TYPE "UDT_VfdSEWPositioningPO"
TITLE = UDT_VFD_SEW_PO
VERSION : 0.1
//User-defined structure of VFD SEW output telegram.
   STRUCT
      Control_Word_1 : Struct   // Control Word 1
         ResetError { ExternalAccessible := 'False'; ExternalVisible := 'False'; ExternalWritable := 'False'} : Bool;   // Reset error "1"
         BIT_09_Reserved { ExternalAccessible := 'False'; ExternalVisible := 'False'; ExternalWritable := 'False'} : Bool;   // Reserved
         ActivateDriveTrain2 { ExternalAccessible := 'False'; ExternalVisible := 'False'; ExternalWritable := 'False'} : Bool;   // Activate drive train 2 "1"
         BIT_11_Reserved { ExternalAccessible := 'False'; ExternalVisible := 'False'; ExternalWritable := 'False'} : Bool;   // Reserved
         DeactivateSW_LimitSwitch { ExternalAccessible := 'False'; ExternalVisible := 'False'; ExternalWritable := 'False'} : Bool;   // Deactivate software limit switch "1"
         ActivateInhibit { ExternalAccessible := 'False'; ExternalVisible := 'False'; ExternalWritable := 'False'} : Bool;   // Activate inhibit "1"
         ActivateStandby { ExternalAccessible := 'False'; ExternalVisible := 'False'; ExternalWritable := 'False'} : Bool;   // Activate standby "1"
         MovikitHandshakeIn { ExternalAccessible := 'False'; ExternalVisible := 'False'; ExternalWritable := 'False'} : Bool;   // If the MOVIKIT works the value will be copied into "MovikitHandshakeOut"
         EnableRapidStop { ExternalAccessible := 'False'; ExternalVisible := 'False'; ExternalWritable := 'False'} : Bool;   // Enable “1” / Rapid stop “0”
         EnableApplicationStop { ExternalAccessible := 'False'; ExternalVisible := 'False'; ExternalWritable := 'False'} : Bool;   // Enable “1” / Application stop “0”
         BIT_02_Reserved { ExternalAccessible := 'False'; ExternalVisible := 'False'; ExternalWritable := 'False'} : Bool;   // Reserved
         ReleaseBrake { ExternalAccessible := 'False'; ExternalVisible := 'False'; ExternalWritable := 'False'} : Bool;   // Release brake "1"
         JogPos { ExternalAccessible := 'False'; ExternalVisible := 'False'; ExternalWritable := 'False'} : Bool;   // Jog in positive direction "1"
         JogNeg { ExternalAccessible := 'False'; ExternalVisible := 'False'; ExternalWritable := 'False'} : Bool;   // Jog in negative direction "1"
         ApplyRelativePositioning { ExternalAccessible := 'False'; ExternalVisible := 'False'; ExternalWritable := 'False'} : Bool;   // Take the relative position from the FCB09 "1"
         StartStop { ExternalAccessible := 'False'; ExternalVisible := 'False'; ExternalWritable := 'False'} : Bool;   // Start "1" / Stop "0"
      END_STRUCT;
      SetpointSpeed : Int;   // Speed (Int) [mm/s]
      SetpointAcceleration : Int;   // Acceleration (Int) [mm/s²]
      SetpointDeceleration : Int;   // Decceleration (Int) [mm/s²]
      DigitalOutputs : Word;   // Digital Outputs
      SetpointMode : Int;   // Set the application mode (Int)
      SetpointPosition_hW : Word;   // Setpoint Position - High Word
      SetpointPosition_lW : Word;   // Setpoint Position - Low Word
   END_STRUCT;

END_TYPE

TYPE "UDT_Message"
TITLE = UDT_Message
VERSION : 0.1
//User-defined structure of the message characters array.
   STRUCT
      Character : Array[0..499] of Char;   // Message character
   END_STRUCT;

END_TYPE

TYPE "UDT_TCPIPReceiveStatistics"
TITLE = UDT_TCPIPReceiveStatistics
VERSION : 0.1
//User-defined structure of FB_TCPIPReceive function block statistics.
   STRUCT
      InvalidMsg : UInt;   // Invalid message received
   END_STRUCT;

END_TYPE

TYPE "UDT_SystemStatistics"
TITLE = Cabinet MCP Statistics
VERSION : 0.1
   STRUCT
      HMI_Stop : "UDT_EventStatistic";   // HMI stop statistics
      Field_Stop : "UDT_EventStatistic";   // Field stop statistics
      Building_EStop : "UDT_EventStatistic";   // Bulding emergency stop statistics
      MCP_EStop : "UDT_EventStatistic";   // MCP emergency stop statistics
      RemotePanel_EStop : "UDT_EventStatistic";   // Remote panel emergency stop statistics
      Error : "UDT_EventStatistic";   // System in error
      StartNumberOfTimes { S7_SetPoint := 'True'} : DInt;   // Number of times system started
      ResetNumberOfTimes { S7_SetPoint := 'True'} : DInt;   // Number of timer system reset
      DataResetNumberOfTimes { S7_SetPoint := 'True'} : DInt;   // Number of data reset
   END_STRUCT;

END_TYPE

TYPE "UDT_ProfiDiagStatistics"
TITLE = UDT_ProfiDiagStatistics
VERSION : 0.1
//User-defined structure of FB_ProfiDiag function block statistics.
   STRUCT
      DeviceError { S7_SetPoint := 'False'} : Array[0..512] of "UDT_EventStatistic";   // Device error statistics
   END_STRUCT;

END_TYPE

TYPE "UDT_PowerDistributionPanelCBState"
VERSION : 0.1
   STRUCT
      CircuitBreakerStateF100 { ExternalAccessible := 'False'; ExternalVisible := 'False'; ExternalWritable := 'False'} : Bool;   // Circuit Breaker State Ok if the signal is true
      CircuitBreakerStateF201 { ExternalAccessible := 'False'; ExternalVisible := 'False'; ExternalWritable := 'False'} : Bool;   // Circuit Breaker State Ok if the signal is true
      CircuitBreakerStateF202 { ExternalAccessible := 'False'; ExternalVisible := 'False'; ExternalWritable := 'False'} : Bool;   // Circuit Breaker State Ok if the signal is true
      CircuitBreakerStateF203 { ExternalAccessible := 'False'; ExternalVisible := 'False'; ExternalWritable := 'False'} : Bool;   // Circuit Breaker State Ok if the signal is true
      CircuitBreakerStateF204 { ExternalAccessible := 'False'; ExternalVisible := 'False'; ExternalWritable := 'False'} : Bool;   // Circuit Breaker State Ok if the signal is true
      CircuitBreakerStateF205 { ExternalAccessible := 'False'; ExternalVisible := 'False'; ExternalWritable := 'False'} : Bool;   // Circuit Breaker State Ok if the signal is true
      CircuitBreakerStateF206 { ExternalAccessible := 'False'; ExternalVisible := 'False'; ExternalWritable := 'False'} : Bool;   // Circuit Breaker State Ok if the signal is true
      CircuitBreakerStateF207 { ExternalAccessible := 'False'; ExternalVisible := 'False'; ExternalWritable := 'False'} : Bool;   // Circuit Breaker State Ok if the signal is true
      CircuitBreakerStateF208 { ExternalAccessible := 'False'; ExternalVisible := 'False'; ExternalWritable := 'False'} : Bool;   // Circuit Breaker State Ok if the signal is true
      CircuitBreakerStateF209 { ExternalAccessible := 'False'; ExternalVisible := 'False'; ExternalWritable := 'False'} : Bool;   // Circuit Breaker State Ok if the signal is true
      CircuitBreakerStateF210 { ExternalAccessible := 'False'; ExternalVisible := 'False'; ExternalWritable := 'False'} : Bool;   // Circuit Breaker State Ok if the signal is true
      CircuitBreakerStateF211 { ExternalAccessible := 'False'; ExternalVisible := 'False'; ExternalWritable := 'False'} : Bool;   // Circuit Breaker State Ok if the signal is true
      CircuitBreakerStateF212 { ExternalAccessible := 'False'; ExternalVisible := 'False'; ExternalWritable := 'False'} : Bool;   // Circuit Breaker State Ok if the signal is true
      CircuitBreakerStateF213 { ExternalAccessible := 'False'; ExternalVisible := 'False'; ExternalWritable := 'False'} : Bool;   // Circuit Breaker State Ok if the signal is true
      CircuitBreakerStateF214 { ExternalAccessible := 'False'; ExternalVisible := 'False'; ExternalWritable := 'False'} : Bool;   // Circuit Breaker State Ok if the signal is true
      CircuitBreakerStateF215 { ExternalAccessible := 'False'; ExternalVisible := 'False'; ExternalWritable := 'False'} : Bool;   // Circuit Breaker State Ok if the signal is true
      CircuitBreakerStateF216 { ExternalAccessible := 'False'; ExternalVisible := 'False'; ExternalWritable := 'False'} : Bool;   // Circuit Breaker State Ok if the signal is true
      CircuitBreakerStateF217 { ExternalAccessible := 'False'; ExternalVisible := 'False'; ExternalWritable := 'False'} : Bool;   // Circuit Breaker State Ok if the signal is true
      CircuitBreakerStateF218 { ExternalAccessible := 'False'; ExternalVisible := 'False'; ExternalWritable := 'False'} : Bool;   // Circuit Breaker State Ok if the signal is true
      CircuitBreakerStateF219 { ExternalAccessible := 'False'; ExternalVisible := 'False'; ExternalWritable := 'False'} : Bool;   // Circuit Breaker State Ok if the signal is true
      CircuitBreakerStateF220 { ExternalAccessible := 'False'; ExternalVisible := 'False'; ExternalWritable := 'False'} : Bool;   // Circuit Breaker State Ok if the signal is true
      CircuitBreakerStateF221 { ExternalAccessible := 'False'; ExternalVisible := 'False'; ExternalWritable := 'False'} : Bool;   // Circuit Breaker State Ok if the signal is true
      CircuitBreakerStateF222 { ExternalAccessible := 'False'; ExternalVisible := 'False'; ExternalWritable := 'False'} : Bool;   // Circuit Breaker State Ok if the signal is true
      CircuitBreakerStateF223 { ExternalAccessible := 'False'; ExternalVisible := 'False'; ExternalWritable := 'False'} : Bool;   // Circuit Breaker State Ok if the signal is true
      CircuitBreakerStateF224 { ExternalAccessible := 'False'; ExternalVisible := 'False'; ExternalWritable := 'False'} : Bool;   // Circuit Breaker State Ok if the signal is true
      CircuitBreakerStateF225 { ExternalAccessible := 'False'; ExternalVisible := 'False'; ExternalWritable := 'False'} : Bool;   // Circuit Breaker State Ok if the signal is true
      CircuitBreakerStateF226 { ExternalAccessible := 'False'; ExternalVisible := 'False'; ExternalWritable := 'False'} : Bool;   // Circuit Breaker State Ok if the signal is true
      CircuitBreakerStateF227 { ExternalAccessible := 'False'; ExternalVisible := 'False'; ExternalWritable := 'False'} : Bool;   // Circuit Breaker State Ok if the signal is true
      CircuitBreakerStateF228 { ExternalAccessible := 'False'; ExternalVisible := 'False'; ExternalWritable := 'False'} : Bool;   // Circuit Breaker State Ok if the signal is true
      CircuitBreakerStateF229 { ExternalAccessible := 'False'; ExternalVisible := 'False'; ExternalWritable := 'False'} : Bool;   // Circuit Breaker State Ok if the signal is true
      CircuitBreakerStateF230 { ExternalAccessible := 'False'; ExternalVisible := 'False'; ExternalWritable := 'False'} : Bool;   // Circuit Breaker State Ok if the signal is true
      CircuitBreakerStateF231 { ExternalAccessible := 'False'; ExternalVisible := 'False'; ExternalWritable := 'False'} : Bool;   // Circuit Breaker State Ok if the signal is true
      CircuitBreakerStateF232 { ExternalAccessible := 'False'; ExternalVisible := 'False'; ExternalWritable := 'False'} : Bool;   // Circuit Breaker State Ok if the signal is true
      CircuitBreakerStateF233 { ExternalAccessible := 'False'; ExternalVisible := 'False'; ExternalWritable := 'False'} : Bool;   // Circuit Breaker State Ok if the signal is true
      CircuitBreakerStateF234 { ExternalAccessible := 'False'; ExternalVisible := 'False'; ExternalWritable := 'False'} : Bool;   // Circuit Breaker State Ok if the signal is true
      CircuitBreakerStateF235 { ExternalAccessible := 'False'; ExternalVisible := 'False'; ExternalWritable := 'False'} : Bool;   // Circuit Breaker State Ok if the signal is true
      CircuitBreakerStateF236 { ExternalAccessible := 'False'; ExternalVisible := 'False'; ExternalWritable := 'False'} : Bool;   // Circuit Breaker State Ok if the signal is true
      CircuitBreakerStateF237 { ExternalAccessible := 'False'; ExternalVisible := 'False'; ExternalWritable := 'False'} : Bool;   // Circuit Breaker State Ok if the signal is true
      CircuitBreakerStateF238 { ExternalAccessible := 'False'; ExternalVisible := 'False'; ExternalWritable := 'False'} : Bool;   // Circuit Breaker State Ok if the signal is true
      CircuitBreakerStateF239 { ExternalAccessible := 'False'; ExternalVisible := 'False'; ExternalWritable := 'False'} : Bool;   // Circuit Breaker State Ok if the signal is true
      CircuitBreakerStateF240 { ExternalAccessible := 'False'; ExternalVisible := 'False'; ExternalWritable := 'False'} : Bool;   // Circuit Breaker State Ok if the signal is true
      CircuitBreakerStateF241 { ExternalAccessible := 'False'; ExternalVisible := 'False'; ExternalWritable := 'False'} : Bool;   // Circuit Breaker State Ok if the signal is true
      CircuitBreakerStateF242 { ExternalAccessible := 'False'; ExternalVisible := 'False'; ExternalWritable := 'False'} : Bool;   // Circuit Breaker State Ok if the signal is true
      CircuitBreakerStateF243 { ExternalAccessible := 'False'; ExternalVisible := 'False'; ExternalWritable := 'False'} : Bool;   // Circuit Breaker State Ok if the signal is true
      CircuitBreakerStateF244 { ExternalAccessible := 'False'; ExternalVisible := 'False'; ExternalWritable := 'False'} : Bool;   // Circuit Breaker State Ok if the signal is true
      CircuitBreakerStateF245 { ExternalAccessible := 'False'; ExternalVisible := 'False'; ExternalWritable := 'False'} : Bool;   // Circuit Breaker State Ok if the signal is true
      CircuitBreakerStateF246 { ExternalAccessible := 'False'; ExternalVisible := 'False'; ExternalWritable := 'False'} : Bool;   // Circuit Breaker State Ok if the signal is true
      CircuitBreakerStateF247 { ExternalAccessible := 'False'; ExternalVisible := 'False'; ExternalWritable := 'False'} : Bool;   // Circuit Breaker State Ok if the signal is true
      CircuitBreakerStateF248 { ExternalAccessible := 'False'; ExternalVisible := 'False'; ExternalWritable := 'False'} : Bool;   // Circuit Breaker State Ok if the signal is true
      CircuitBreakerStateF249 { ExternalAccessible := 'False'; ExternalVisible := 'False'; ExternalWritable := 'False'} : Bool;   // Circuit Breaker State Ok if the signal is true
      CircuitBreakerStateF250 { ExternalAccessible := 'False'; ExternalVisible := 'False'; ExternalWritable := 'False'} : Bool;   // Circuit Breaker State Ok if the signal is true
      CircuitBreakerStateF251 { ExternalAccessible := 'False'; ExternalVisible := 'False'; ExternalWritable := 'False'} : Bool;   // Circuit Breaker State Ok if the signal is true
      CircuitBreakerStateF501 { ExternalAccessible := 'False'; ExternalVisible := 'False'; ExternalWritable := 'False'} : Bool;   // Circuit Breaker State Ok if the signal is true
      CircuitBreakerStateF502 { ExternalAccessible := 'False'; ExternalVisible := 'False'; ExternalWritable := 'False'} : Bool;   // Circuit Breaker State Ok if the signal is true
      CircuitBreakerStateF503 { ExternalAccessible := 'False'; ExternalVisible := 'False'; ExternalWritable := 'False'} : Bool;   // Circuit Breaker State Ok if the signal is true
      CircuitBreakerStateF504 { ExternalAccessible := 'False'; ExternalVisible := 'False'; ExternalWritable := 'False'} : Bool;   // Circuit Breaker State Ok if the signal is true
      CircuitBreakerStateF505 { ExternalAccessible := 'False'; ExternalVisible := 'False'; ExternalWritable := 'False'} : Bool;   // Circuit Breaker State Ok if the signal is true
   END_STRUCT;

END_TYPE

TYPE "UDT_PowerDistributionPanelStatus"
VERSION : 0.1
   STRUCT
      Status : Int;   // Status number
      Specific : Struct
         CircuitBreakersTripped { ExternalAccessible := 'False'; ExternalVisible := 'False'; ExternalWritable := 'False'} : Bool;   // Circuit breakers tripped when the value is true
         CircuitBreakerTrippedF100 { ExternalAccessible := 'False'; ExternalVisible := 'False'; ExternalWritable := 'False'} : Bool;   // Circuit breaker is tripped when the value is true
         CircuitBreakerTrippedF201 { ExternalAccessible := 'False'; ExternalVisible := 'False'; ExternalWritable := 'False'} : Bool;   // Circuit breaker is tripped when the value is true
         CircuitBreakerTrippedF202 { ExternalAccessible := 'False'; ExternalVisible := 'False'; ExternalWritable := 'False'} : Bool;   // Circuit breaker is tripped when the value is true
         CircuitBreakerTrippedF203 { ExternalAccessible := 'False'; ExternalVisible := 'False'; ExternalWritable := 'False'} : Bool;   // Circuit breaker is tripped when the value is true
         CircuitBreakerTrippedF204 { ExternalAccessible := 'False'; ExternalVisible := 'False'; ExternalWritable := 'False'} : Bool;   // Circuit breaker is tripped when the value is true
         CircuitBreakerTrippedF205 { ExternalAccessible := 'False'; ExternalVisible := 'False'; ExternalWritable := 'False'} : Bool;   // Circuit breaker is tripped when the value is true
         CircuitBreakerTrippedF206 { ExternalAccessible := 'False'; ExternalVisible := 'False'; ExternalWritable := 'False'} : Bool;   // Circuit breaker is tripped when the value is true
         CircuitBreakerTrippedF207 { ExternalAccessible := 'False'; ExternalVisible := 'False'; ExternalWritable := 'False'} : Bool;   // Circuit breaker is tripped when the value is true
         CircuitBreakerTrippedF208 { ExternalAccessible := 'False'; ExternalVisible := 'False'; ExternalWritable := 'False'} : Bool;   // Circuit breaker is tripped when the value is true
         CircuitBreakerTrippedF209 { ExternalAccessible := 'False'; ExternalVisible := 'False'; ExternalWritable := 'False'} : Bool;   // Circuit breaker is tripped when the value is true
         CircuitBreakerTrippedF210 { ExternalAccessible := 'False'; ExternalVisible := 'False'; ExternalWritable := 'False'} : Bool;   // Circuit breaker is tripped when the value is true
         CircuitBreakerTrippedF211 { ExternalAccessible := 'False'; ExternalVisible := 'False'; ExternalWritable := 'False'} : Bool;   // Circuit breaker is tripped when the value is true
         CircuitBreakerTrippedF212 { ExternalAccessible := 'False'; ExternalVisible := 'False'; ExternalWritable := 'False'} : Bool;   // Circuit breaker is tripped when the value is true
         CircuitBreakerTrippedF213 { ExternalAccessible := 'False'; ExternalVisible := 'False'; ExternalWritable := 'False'} : Bool;   // Circuit breaker is tripped when the value is true
         CircuitBreakerTrippedF214 { ExternalAccessible := 'False'; ExternalVisible := 'False'; ExternalWritable := 'False'} : Bool;   // Circuit breaker is tripped when the value is true
         CircuitBreakerTrippedF215 { ExternalAccessible := 'False'; ExternalVisible := 'False'; ExternalWritable := 'False'} : Bool;   // Circuit breaker is tripped when the value is true
         CircuitBreakerTrippedF216 { ExternalAccessible := 'False'; ExternalVisible := 'False'; ExternalWritable := 'False'} : Bool;   // Circuit breaker is tripped when the value is true
         CircuitBreakerTrippedF217 { ExternalAccessible := 'False'; ExternalVisible := 'False'; ExternalWritable := 'False'} : Bool;   // Circuit breaker is tripped when the value is true
         CircuitBreakerTrippedF218 { ExternalAccessible := 'False'; ExternalVisible := 'False'; ExternalWritable := 'False'} : Bool;   // Circuit breaker is tripped when the value is true
         CircuitBreakerTrippedF219 { ExternalAccessible := 'False'; ExternalVisible := 'False'; ExternalWritable := 'False'} : Bool;   // Circuit breaker is tripped when the value is true
         CircuitBreakerTrippedF220 { ExternalAccessible := 'False'; ExternalVisible := 'False'; ExternalWritable := 'False'} : Bool;   // Circuit breaker is tripped when the value is true
         CircuitBreakerTrippedF221 { ExternalAccessible := 'False'; ExternalVisible := 'False'; ExternalWritable := 'False'} : Bool;   // Circuit breaker is tripped when the value is true
         CircuitBreakerTrippedF222 { ExternalAccessible := 'False'; ExternalVisible := 'False'; ExternalWritable := 'False'} : Bool;   // Circuit breaker is tripped when the value is true
         CircuitBreakerTrippedF223 { ExternalAccessible := 'False'; ExternalVisible := 'False'; ExternalWritable := 'False'} : Bool;   // Circuit breaker is tripped when the value is true
         CircuitBreakerTrippedF224 { ExternalAccessible := 'False'; ExternalVisible := 'False'; ExternalWritable := 'False'} : Bool;   // Circuit breaker is tripped when the value is true
         CircuitBreakerTrippedF225 { ExternalAccessible := 'False'; ExternalVisible := 'False'; ExternalWritable := 'False'} : Bool;   // Circuit breaker is tripped when the value is true
         CircuitBreakerTrippedF226 { ExternalAccessible := 'False'; ExternalVisible := 'False'; ExternalWritable := 'False'} : Bool;   // Circuit breaker is tripped when the value is true
         CircuitBreakerTrippedF227 { ExternalAccessible := 'False'; ExternalVisible := 'False'; ExternalWritable := 'False'} : Bool;   // Circuit breaker is tripped when the value is true
         CircuitBreakerTrippedF228 { ExternalAccessible := 'False'; ExternalVisible := 'False'; ExternalWritable := 'False'} : Bool;   // Circuit breaker is tripped when the value is true
         CircuitBreakerTrippedF229 { ExternalAccessible := 'False'; ExternalVisible := 'False'; ExternalWritable := 'False'} : Bool;   // Circuit breaker is tripped when the value is true
         CircuitBreakerTrippedF230 { ExternalAccessible := 'False'; ExternalVisible := 'False'; ExternalWritable := 'False'} : Bool;   // Circuit breaker is tripped when the value is true
         CircuitBreakerTrippedF231 { ExternalAccessible := 'False'; ExternalVisible := 'False'; ExternalWritable := 'False'} : Bool;   // Circuit breaker is tripped when the value is true
         CircuitBreakerTrippedF232 { ExternalAccessible := 'False'; ExternalVisible := 'False'; ExternalWritable := 'False'} : Bool;   // Circuit breaker is tripped when the value is true
         CircuitBreakerTrippedF233 { ExternalAccessible := 'False'; ExternalVisible := 'False'; ExternalWritable := 'False'} : Bool;   // Circuit breaker is tripped when the value is true
         CircuitBreakerTrippedF234 { ExternalAccessible := 'False'; ExternalVisible := 'False'; ExternalWritable := 'False'} : Bool;   // Circuit breaker is tripped when the value is true
         CircuitBreakerTrippedF235 { ExternalAccessible := 'False'; ExternalVisible := 'False'; ExternalWritable := 'False'} : Bool;   // Circuit breaker is tripped when the value is true
         CircuitBreakerTrippedF236 { ExternalAccessible := 'False'; ExternalVisible := 'False'; ExternalWritable := 'False'} : Bool;   // Circuit breaker is tripped when the value is true
         CircuitBreakerTrippedF237 { ExternalAccessible := 'False'; ExternalVisible := 'False'; ExternalWritable := 'False'} : Bool;   // Circuit breaker is tripped when the value is true
         CircuitBreakerTrippedF238 { ExternalAccessible := 'False'; ExternalVisible := 'False'; ExternalWritable := 'False'} : Bool;   // Circuit breaker is tripped when the value is true
         CircuitBreakerTrippedF239 { ExternalAccessible := 'False'; ExternalVisible := 'False'; ExternalWritable := 'False'} : Bool;   // Circuit breaker is tripped when the value is true
         CircuitBreakerTrippedF240 { ExternalAccessible := 'False'; ExternalVisible := 'False'; ExternalWritable := 'False'} : Bool;   // Circuit breaker is tripped when the value is true
         CircuitBreakerTrippedF241 { ExternalAccessible := 'False'; ExternalVisible := 'False'; ExternalWritable := 'False'} : Bool;   // Circuit breaker is tripped when the value is true
         CircuitBreakerTrippedF242 { ExternalAccessible := 'False'; ExternalVisible := 'False'; ExternalWritable := 'False'} : Bool;   // Circuit breaker is tripped when the value is true
         CircuitBreakerTrippedF243 { ExternalAccessible := 'False'; ExternalVisible := 'False'; ExternalWritable := 'False'} : Bool;   // Circuit breaker is tripped when the value is true
         CircuitBreakerTrippedF244 { ExternalAccessible := 'False'; ExternalVisible := 'False'; ExternalWritable := 'False'} : Bool;   // Circuit breaker is tripped when the value is true
         CircuitBreakerTrippedF245 { ExternalAccessible := 'False'; ExternalVisible := 'False'; ExternalWritable := 'False'} : Bool;   // Circuit breaker is tripped when the value is true
         CircuitBreakerTrippedF246 { ExternalAccessible := 'False'; ExternalVisible := 'False'; ExternalWritable := 'False'} : Bool;   // Circuit breaker is tripped when the value is true
         CircuitBreakerTrippedF247 { ExternalAccessible := 'False'; ExternalVisible := 'False'; ExternalWritable := 'False'} : Bool;   // Circuit breaker is tripped when the value is true
         CircuitBreakerTrippedF248 { ExternalAccessible := 'False'; ExternalVisible := 'False'; ExternalWritable := 'False'} : Bool;   // Circuit breaker is tripped when the value is true
         CircuitBreakerTrippedF249 { ExternalAccessible := 'False'; ExternalVisible := 'False'; ExternalWritable := 'False'} : Bool;   // Circuit breaker is tripped when the value is true
         CircuitBreakerTrippedF250 { ExternalAccessible := 'False'; ExternalVisible := 'False'; ExternalWritable := 'False'} : Bool;   // Circuit breaker is tripped when the value is true
         CircuitBreakerTrippedF501 { ExternalAccessible := 'False'; ExternalVisible := 'False'; ExternalWritable := 'False'} : Bool;   // Circuit breaker is tripped when the value is true
         CircuitBreakerTrippedF502 { ExternalAccessible := 'False'; ExternalVisible := 'False'; ExternalWritable := 'False'} : Bool;   // Circuit breaker is tripped when the value is true
         CircuitBreakerTrippedF503 { ExternalAccessible := 'False'; ExternalVisible := 'False'; ExternalWritable := 'False'} : Bool;   // Circuit breaker is tripped when the value is true
         CircuitBreakerTrippedF504 { ExternalAccessible := 'False'; ExternalVisible := 'False'; ExternalWritable := 'False'} : Bool;   // Circuit breaker is tripped when the value is true
         CircuitBreakerTrippedF505 { ExternalAccessible := 'False'; ExternalVisible := 'False'; ExternalWritable := 'False'} : Bool;   // Circuit breaker is tripped when the value is true
      END_STRUCT;
   END_STRUCT;

END_TYPE

TYPE "UDT_XBSInductInterfaceRcv"
VERSION : 0.1
   STRUCT
      Watchdog : Byte;   // Watchdog counter
      RunConsent { ExternalAccessible := 'False'; ExternalVisible := 'False'; ExternalWritable := 'False'} : Bool;   // Ready to receive
      Running { ExternalAccessible := 'False'; ExternalVisible := 'False'; ExternalWritable := 'False'} : Bool;   // The IDS is moving
      Fault { ExternalAccessible := 'False'; ExternalVisible := 'False'; ExternalWritable := 'False'} : Bool;   // The IDS is in fault status
      Enabled { ExternalAccessible := 'False'; ExternalVisible := 'False'; ExternalWritable := 'False'} : Bool;   // The IDS is allowed to laod packages on Sorter
      Throughput : DInt;   // Production target
      LastConveyorSpeedSP : Real;   // Maximum Speed setpoint for the last conveyor of the upstream line (mm/sec)
      MinimumGap : Real;   // Minimum gap between the head and the tail of parcels
   END_STRUCT;

END_TYPE

TYPE "UDT_InchingConfiguration"
TITLE = UDT_InchingConfiguration
VERSION : 0.1
//User-defined structure of inching block parameters.
   STRUCT
      GapSize : Int;   // Gapsize in [cm]
      MaximalFillingPosition : Int;   // Position in [cm] from the end
      ButtonReleaseDelayTime : UDInt;   // Time in [ms] to accept the button to set full or release
      WaitForStartConf { ExternalAccessible := 'False'; ExternalVisible := 'False'; ExternalWritable := 'False'} : Bool;   // True = Wait for conformation to start after running empty
   END_STRUCT;

END_TYPE

TYPE "UDT_VfdSiemensPO"
TITLE = UDT_VFD_Siemens_PO
VERSION : 0.1
//User-defined structure of VFD Siemens output telegram.
   STRUCT
      STW_1 : Struct   // Control Word Interconnection 1
         ForceDormantErrorTest { ExternalAccessible := 'False'; ExternalVisible := 'False'; ExternalWritable := 'False'} : Bool;   // Only applicable in G120 with safety motion monitoring
         SpareBit9 { ExternalAccessible := 'False'; ExternalVisible := 'False'; ExternalWritable := 'False'} : Bool;   // Spare bit 9
         ControlViaPLC { ExternalAccessible := 'False'; ExternalVisible := 'False'; ExternalWritable := 'False'} : Bool;   // 1 = Control via PLC (Control via fieldbus, inverter accepts the process data from the fieldbus), 0 = No control via PLC (Inverter ignores the process data from the fieldbus) p 0854[0] = r 2090.10
         DirectionReversal { ExternalAccessible := 'False'; ExternalVisible := 'False'; ExternalWritable := 'False'} : Bool;   // 0 = Direction reversal (Invert setpoint of the inverter) p1113[0] = r 2090.11
         SpareBit12 { ExternalAccessible := 'False'; ExternalVisible := 'False'; ExternalWritable := 'False'} : Bool;   // Spare bit 12
         SpareBit13 { ExternalAccessible := 'False'; ExternalVisible := 'False'; ExternalWritable := 'False'} : Bool;   // Spare bit 13
         SpareBit14 { ExternalAccessible := 'False'; ExternalVisible := 'False'; ExternalWritable := 'False'} : Bool;   // Spare bit 14
         SpareBit15 { ExternalAccessible := 'False'; ExternalVisible := 'False'; ExternalWritable := 'False'} : Bool;   // Spare bit 15
         ONOFF1 { ExternalAccessible := 'False'; ExternalVisible := 'False'; ExternalWritable := 'False'} : Bool;   // 0 --> 1 = ON (The inverter goes to "ready "state. If, in addition bit 3 = 1 then the inverter switches on the motor), 0 = OFF1 (The motor brakes with ramp-down time p1121 of the ramp-function generator. The inverter switches off the motor an standstill) p0840[0] = r 2090.0
         OFF2 { ExternalAccessible := 'False'; ExternalVisible := 'False'; ExternalWritable := 'False'} : Bool;   // 1 = No OFF2 (The motor can be switched on (ON command)), 0 = OFF2 (Switch off the motor immediately, the motor then coasts down to a standstill) p0844[0] = r 2090.1
         OFF3 { ExternalAccessible := 'False'; ExternalVisible := 'False'; ExternalWritable := 'False'} : Bool;   // 1 = No OFF3 (The motor can be switched on (ON command)), 0 = OFF3 (Quick stop: The motor brakes with the OFF3 ramp-down time p 1135 down to a standstill.) p0848[0] = r 2090.2
         EnableOperation { ExternalAccessible := 'False'; ExternalVisible := 'False'; ExternalWritable := 'False'} : Bool;   // 1 = Enable operation (Switch on motor (pulses can be enabled)), 0 = Inhibit operation (Immediately switch off motor (cancel pulses)) p 0852[0] = r 2090.3
         DoNotDisableRFG { ExternalAccessible := 'False'; ExternalVisible := 'False'; ExternalWritable := 'False'} : Bool;   // 1 = Do not disable RFG (The ramp-function generator can be enabled), 0 = Disable RFG (The inverter immedeately sets its ramp-function generator output to 0) p 1140[0] = r 2090.4
         EnableRFG { ExternalAccessible := 'False'; ExternalVisible := 'False'; ExternalWritable := 'False'} : Bool;   // 1 = Enable RFG (The output of the ramp-function generator follows the setpoint), 0 = Stop RFG (The output of the ramp-function generator stops at the actual value) p1141[0] = r 2090.5
         EnableSetpoint { ExternalAccessible := 'False'; ExternalVisible := 'False'; ExternalWritable := 'False'} : Bool;   // 1 = Enable setpoint (Motor accelerates with the ramp-up time p1120 to the setpoint), 0 = Inhibit setpoint (The inverter brakes the motor with the ramp-down time p1121 of the ramp-function generator) p 1142[0] = r 2090.6
         Acknowledge { ExternalAccessible := 'False'; ExternalVisible := 'False'; ExternalWritable := 'False'} : Bool;   // 0 --> 1 = Acknowledge faults (Acknowledge fault. If the ON command is still active, the inverter switches to "closing lockout" state) p 2103[0] = r 2090.7
      END_STRUCT;
      SpeedSetpoint : Int;   // Speed Setpoint 100%=4000 HEX = 16384 DEZnormalisation with p 2000 of the inverter
      SetpointAcceleration : Int;   // Acceleration time, defalut time scale in VFD in the rage 0...200%=0...7FFF HEX= 0...32767
      SetpointDeceleration : Int;   // Decceleration time, defalut time scale in VFD in the rage 0...200%=0...7FFF HEX= 0...32767
      SpareWord5 : Int;   // Spare Word 5
      SpareWord6 : Int;   // Spare Word 6
      SpareWord7 : Int;   // Spare Word 7
      SpareWord8 : Int;   // Spare Word 8
      SpareWord9 : Int;   // Spare Word 9
      SpareWord10 : Int;   // Spare Word 10
      SpareWord11 : Int;   // Spare Word 11
   END_STRUCT;

END_TYPE

TYPE "UDT_UnloaderConfiguration"
TITLE = UDT_UnloaderConfiguration
VERSION : 0.1
//User-defined structure of unloader parameters.
   STRUCT
      PEC_EOS : "UDT_PECConfiguration";   // Photo eye time on delay
      Speedsetpoint : Int;   // Speedsetpoint: 0=Low, 1=Nom, 2=High
      EnergySaveLength : Int;   // Distance conveyor travelled before energy save activate [cm]
      FirstConveyorToStart { ExternalAccessible := 'False'; ExternalVisible := 'False'; ExternalWritable := 'False'} : Bool;   // First conveyor to start cascade mode
      Energy { ExternalAccessible := 'False'; ExternalVisible := 'False'; ExternalWritable := 'False'} : Bool;   // Energy save mode enable
   END_STRUCT;

END_TYPE

TYPE "UDT_UnloaderStatistics"
TITLE = UDT_UnloaderStatistics
VERSION : 0.1
//User-defined structure of FB_Unloader function block statistics.
   STRUCT
      EnergySave : "UDT_EventStatistic";   // Number of times that save energy mode occurs
      ExtendableUpTime : "UDT_EventStatistic";   // Conveyor up time
      ExtendableDownTime : "UDT_EventStatistic";   // Conveyor down time
      VFDError : "UDT_EventStatistic";   // VFD Error
      NotHealthy : "UDT_EventStatistic";   // Extendable not healthy
      TooLongParcel : "UDT_EventStatistic";   // Too long parcels
      PEC_EOS : "UDT_PECStatistics";   // PEC error
   END_STRUCT;

END_TYPE

TYPE "UDT_Connection"
TITLE = UDT_Connection
VERSION : 0.1
//User-defined structure of connection parameters.
   STRUCT
      ActiveEstablished : Bool := FALSE;   // 0 – Passive connection establishment; 1 – Active connection establishment
      Interface_ID : HW_ANY := 64;   // Interface ID of CPU Ethernet interface
      ID : CONN_OUC;   // Unique ID as system reference for the connection
      IP : Array[1..4] of Int;   // IP address
      Port : UInt;   // Port number of the communication partner
      ConTimeout : DInt;   // Maximum waiting time for response from the communication partner [ms]
   END_STRUCT;

END_TYPE

TYPE "UDT_TCPIPConnectStatus"
TITLE = UDT_TCPIPConnectStatus
VERSION : 0.1
//User-defined structure of FB_TCPIPConnect function block status.
   STRUCT
      Status : Int;   // Status number
      Specific : Struct   // Specific status structure
         ErrorCode : Struct   // Error code structure
            TCON : Word;   // Siemens TCON error code - Check documetation
            TDISCON : Word;   // Siemens TDISCON error code - Check documetation
            TDIAG : Word;   // Siemens TDIAG error code - Check documetation
         END_STRUCT;
         Connected { ExternalAccessible := 'False'; ExternalVisible := 'False'; ExternalWritable := 'False'} : Bool;   // Connected
         CommunicationFault { ExternalAccessible := 'False'; ExternalVisible := 'False'; ExternalWritable := 'False'} : Bool;   // Communication fault
      END_STRUCT;
   END_STRUCT;

END_TYPE

TYPE "UDT_TCPIPConnectStatistics"
TITLE = UDT_TCPIPConnectStatistics
VERSION : 0.1
//User-defined structure of FB_TCPIPConnect function block statistics.
   STRUCT
      ConnectionLost { S7_SetPoint := 'False'} : "UDT_EventStatistic";   // Connection lost statistics
   END_STRUCT;

END_TYPE

TYPE "UDT_SystemControlStatus"
TITLE = UDT_SystemControlStatus
VERSION : 0.1
//User-defined structure of FB_SystemControl function block status.
   STRUCT
      Status : Int;   // Status number
   END_STRUCT;

END_TYPE

TYPE "UDT_SystemControlCommand"
TITLE = UDT_SystemControlCommand
VERSION : 0.1
//User-defined structure of system control commands.
   STRUCT
      Start { ExternalAccessible := 'False'; ExternalVisible := 'False'; ExternalWritable := 'False'} : Bool;   // Start Command from HMI
      Stop { ExternalAccessible := 'False'; ExternalVisible := 'False'; ExternalWritable := 'False'} : Bool;   // Stop command from HMI
      Reset { ExternalAccessible := 'False'; ExternalVisible := 'False'; ExternalWritable := 'False'} : Bool;   // Reset command from HMI
      ResetData { ExternalAccessible := 'False'; ExternalVisible := 'False'; ExternalWritable := 'False'} : Bool;   // Reset data command from HMI
      ResetSafety { ExternalAccessible := 'False'; ExternalVisible := 'False'; ExternalWritable := 'False'} : Bool;   // Reset safety command from HMI
      ManualMode { ExternalAccessible := 'False'; ExternalVisible := 'False'; ExternalWritable := 'False'} : Bool;   // Manual mode command from HMI
   END_STRUCT;

END_TYPE

TYPE "UDT_SystemControlStatistics"
TITLE = UDT_SystemControlStatistics
VERSION : 0.1
//User-defined structure of FB_SystemControl function block statistics.
   STRUCT
      Run : "UDT_EventStatistic";   // Equipment run statistics
      Error : "UDT_EventStatistic";   // Equipment error statistics
      EnergySave : "UDT_EventStatistic";   // Equipment energy save statistics
   END_STRUCT;

END_TYPE

TYPE "UDT_MainControlPanelStatistics"
TITLE = Cabinet MCP Statistics
VERSION : 0.1
   STRUCT
      UPSFault : "UDT_EventStatistic";   // Unit Power Supply fault statistics
      FireAlarm : "UDT_EventStatistic";   // Fire Alarm active statistics
      "230VAC_CB101F1Tripped" : "UDT_EventStatistic";   // Circuit braker 101F1 tripped  statistics
      "230VAC_CB101F4Tripped" : "UDT_EventStatistic";   // Circuit braker 101F4 tripped statistics
      "230VAC_CB102F1Tripped" : "UDT_EventStatistic";   // Circuit braker 102F1 tripped statistics
      "230VAC_CB102F3Tripped" : "UDT_EventStatistic";   // Circuit braker 102F3 tripped statistics
      "230VAC_CB201F4Tripped" : "UDT_EventStatistic";   // Circuit braker 201F4 tripped statistics
      "24VDC_CB201F1Tripped" : "UDT_EventStatistic";   // Circuit braker 201F1 tripped statistics
      "24VDC_CB205F5Tripped" : "UDT_EventStatistic";   // Circuit braker 205F5 tripped statistics
      "24VDC_CB205F9Tripped" : "UDT_EventStatistic";   // Circuit braker 205F9 tripped statistics
      ScalanceSwitchStatus : "UDT_EventStatistic";   // Scalance switch status statistics
      Spare_1 : "UDT_EventStatistic";   // Spare
      Spare_2 : "UDT_EventStatistic";   // Spare
      Spare_3 : "UDT_EventStatistic";   // Spare
      PS_201T1_Tripped { S7_SetPoint := 'False'} : "UDT_EventStatistic";   // Circuit braker 201T1 tripped statistics
      "PN/PNCouplerFault" : "UDT_EventStatistic";   // PN/PN coupler fault statistics
      SingulatorCouplerFault : "UDT_EventStatistic";   // ProSoft coupler fault statistics
      ScalanceSwitchFault : "UDT_EventStatistic";   // Scalance switch fault statistics
      IOModuleCouplerFault : "UDT_EventStatistic";   // IO Module fault statistics
      RackModuleFault : "UDT_EventStatistic";   // A module fault occurred in the mainrack
   END_STRUCT;

END_TYPE

TYPE "UDT_MainControlPanelStatus"
TITLE = Cabinet MCP Status
VERSION : 0.1
   STRUCT
      Status : Int;   //  Status number
      Specific : Struct
         PN_PN_MSP_PNSlaveNotOnline { ExternalAccessible := 'False'; ExternalVisible := 'False'; ExternalWritable := 'False'} : Bool;   //  PNPN coupler is not online
         PN_PN_MSP_PNSlaveError { ExternalAccessible := 'False'; ExternalVisible := 'False'; ExternalWritable := 'False'} : Bool;   //  PNPN coupler has an error
         PN_PN_MSP_PNSlaveWarning { ExternalAccessible := 'False'; ExternalVisible := 'False'; ExternalWritable := 'False'} : Bool;   //  PNPN coupler has a warning
         IOModule_PNSlaveNotOnline { ExternalAccessible := 'False'; ExternalVisible := 'False'; ExternalWritable := 'False'} : Bool;   // I/O Module is not online
         IOModule_PNSlaveError { ExternalAccessible := 'False'; ExternalVisible := 'False'; ExternalWritable := 'False'} : Bool;   // I/O Module has an error
         IOModule_PNSlaveWarning { ExternalAccessible := 'False'; ExternalVisible := 'False'; ExternalWritable := 'False'} : Bool;   // I/O Module has a warning
         ScalanceSwitchPNSlaveNotOnline { ExternalAccessible := 'False'; ExternalVisible := 'False'; ExternalWritable := 'False'} : Bool;   // Scalance switch is not online
         ScalanceSwitchPNSlaveError { ExternalAccessible := 'False'; ExternalVisible := 'False'; ExternalWritable := 'False'} : Bool;   // Scalance switch has an error
         ScalanceSwitchPNSlaveWarning { ExternalAccessible := 'False'; ExternalVisible := 'False'; ExternalWritable := 'False'} : Bool;   // Scalance switch has a warning
         ScalanceSwitchStatus { ExternalAccessible := 'False'; ExternalVisible := 'False'; ExternalWritable := 'False'} : Bool;   // TRUE when Scalance switch is not healthy
         Singulator_PNSlaveNotOnline { ExternalAccessible := 'False'; ExternalVisible := 'False'; ExternalWritable := 'False'} : Bool;   // Singulator coupler is not online
         Singulator_PNSlaveError { ExternalAccessible := 'False'; ExternalVisible := 'False'; ExternalWritable := 'False'} : Bool;   // Singulator coupler has an error
         Singulator_PNSlaveWarning { ExternalAccessible := 'False'; ExternalVisible := 'False'; ExternalWritable := 'False'} : Bool;   // Singulator coupler has a warning
         UPSSwitchTripped { ExternalAccessible := 'False'; ExternalVisible := 'False'; ExternalWritable := 'False'} : Bool;   //  Unit Power Supply switch tripped
         FireAlarmActive { ExternalAccessible := 'False'; ExternalVisible := 'False'; ExternalWritable := 'False'} : Bool;   //  Fire alarm active when the signal is true
         PS_201T1_Tripped { ExternalAccessible := 'False'; ExternalVisible := 'False'; ExternalWritable := 'False'} : Bool;   //  TRUE if power supply 201T1 tripped
         "230VAC_CB201F4Tripped" { ExternalAccessible := 'False'; ExternalVisible := 'False'; ExternalWritable := 'False'} : Bool;   //  TRUE if MCP circuit breaker 201F4 tripped
         "230VAC_CB101F1Tripped" { ExternalAccessible := 'False'; ExternalVisible := 'False'; ExternalWritable := 'False'} : Bool;   //  TRUE if MCP circuit breaker 101F1 tripped
         "230VAC_CB101F4Tripped" { ExternalAccessible := 'False'; ExternalVisible := 'False'; ExternalWritable := 'False'} : Bool;   //  TRUE if MCP circuit breaker 101F4 tripped
         "230VAC_CB102F1Tripped" { ExternalAccessible := 'False'; ExternalVisible := 'False'; ExternalWritable := 'False'} : Bool;   //  TRUE if MCU circuit breaker 102F1 tripped
         "230VAC_CB102F3Tripped" { ExternalAccessible := 'False'; ExternalVisible := 'False'; ExternalWritable := 'False'} : Bool;   //  TRUE if MCU circuit breaker 102F3 tripped
         "24VDC_CB201F1Tripped" { ExternalAccessible := 'False'; ExternalVisible := 'False'; ExternalWritable := 'False'} : Bool;   //  TRUE if MCU circuit breaker 205F1 tripped
         "24VDC_CB205F5Tripped" { ExternalAccessible := 'False'; ExternalVisible := 'False'; ExternalWritable := 'False'} : Bool;   //  TRUE if MCU circuit breaker 205F5 tripped
         "24VDC_CB205F9Tripped" { ExternalAccessible := 'False'; ExternalVisible := 'False'; ExternalWritable := 'False'} : Bool;   //  TRUE if MCU circuit breaker 205F9 tripped
         Spare_1 { ExternalAccessible := 'False'; ExternalVisible := 'False'; ExternalWritable := 'False'} : Bool;   // Spare
         Spare_2 { ExternalAccessible := 'False'; ExternalVisible := 'False'; ExternalWritable := 'False'} : Bool;   // Spare
         Spare_3 { ExternalAccessible := 'False'; ExternalVisible := 'False'; ExternalWritable := 'False'} : Bool;   // Spare
         RackSlotError : Array[0..31] of Bool;   //  One of the main rack slots has an error
         IOModuleSlotError : Array[0..31] of Bool;   //  Module error
      END_STRUCT;
   END_STRUCT;

END_TYPE

TYPE "UDT_StopRollerConfiguration"
VERSION : 0.1
   STRUCT
      BrakePuls : UDInt;   // Time [ms] brake is up in brake function
      BrakePause : UDInt;   // Time [ms] brake is down in brake function
      BrakePauseLong : UDInt;   // Long time [ms] brake is down in brake function
      PECBrakeOnDelay : UDInt;   // On delay time PEC brake signal
      PECBrakeOffDelay : UDInt;   // Off delay time PEC brake signal
      PECStopOnDelay : UDInt;   // On delay time PEC stop signal
      PECStopOffDelay : UDInt;   // Off delay time PEC stop signal
      StopFunctionOnDelay : UDInt;   // On delay time stop function
      StopFunctionOffDelay : UDInt;   // Off delay time stop function
      FailSafe { ExternalAccessible := 'False'; ExternalVisible := 'False'; ExternalWritable := 'False'} : Bool;   // Activate output to release
   END_STRUCT;

END_TYPE

FUNCTION_BLOCK "FB_AMBASpiralSlatCheck"
{ S7_Optimized_Access := 'TRUE' }
VERSION : 0.1
// ATTRIBUTES
// AUTO_NUMBER = True
// BLOCK_NUMBER = 254
// END_ATTRIBUTES
   VAR_INPUT
      ix_SlatDetection { ExternalAccessible := 'False'; ExternalVisible := 'False'; ExternalWritable := 'False'} : Bool;   // Proximity switch signal (TRUE = Slat detected)
      ix_HardwareOk { ExternalAccessible := 'False'; ExternalVisible := 'False'; ExternalWritable := 'False'} : Bool;   // TRUE when hardware is Ok
   END_VAR

   VAR_IN_OUT
      iqx_MissingSlatDetected { ExternalAccessible := 'False'; ExternalVisible := 'False'; ExternalWritable := 'False'} : Bool;   // [Failure] Missing slat detected (TRUE = detected)
      iqUDT_Statistics : "UDT_EventStatistic";   // Statistics of missing slat
      iqUDT_EquipmentControl : "UDT_EquipmentControl";
   END_VAR

   VAR
      sFB_SignalFilter { ExternalAccessible := 'False'; ExternalVisible := 'False'; ExternalWritable := 'False'; S7_SetPoint := 'False'} : "FB_TimerOnOffDelay";   // On/Off delay to filter the input signal
      sR_TRIG_MissingSlatDetected {InstructionName := 'R_TRIG'; LibVersion := '1.0'; ExternalAccessible := 'False'; ExternalVisible := 'False'; ExternalWritable := 'False'; S7_SetPoint := 'False'} : R_TRIG;   // Flank detection missing slat
   END_VAR

   VAR_TEMP
      tx_SlatDetected : Bool;
   END_VAR

   VAR CONSTANT
      cudi_OffDelay : UDInt := 25;   // [ms]
   END_VAR


BEGIN
	(*
	Version history:
	Date        | Version   | Author              | Remark
	----------------------------------------------------------------------------------------
	 14/03/2022 | 1.0       | G.Vlooswijk         | Initial version for FedEx Milano
	 16/05/2022 | 1.1       | G.Vlooswijk         | Tested (logic) GLS Tongeren
	 03/06/2024 | 1.2       | J.Majer             | Adapted to current library
	*)

	REGION Inputs

	    // Filter input signal
	    #sFB_SignalFilter(iudi_OffDelayTime := #cudi_OffDelay,
	                      ix_SignalToDelay := #ix_SlatDetection,
	                      qx_DelayedSignal => #tx_SlatDetected);

	END_REGION

	REGION Missing slat detection

	    //Set fault
	    IF NOT #tx_SlatDetected AND #ix_HardwareOk THEN
	        #iqx_MissingSlatDetected := TRUE;
	    END_IF;

	    //Reset fault
	    IF #iqx_MissingSlatDetected
	        AND (NOT #ix_HardwareOk
	        OR #tx_SlatDetected AND #iqUDT_EquipmentControl.Command.Reset)
	    THEN
	        #iqx_MissingSlatDetected := FALSE;
	    END_IF;

	END_REGION

	REGION Statistics

	    // Rising flank detection
	    #sR_TRIG_MissingSlatDetected(CLK := #iqx_MissingSlatDetected);

	    IF #iqx_MissingSlatDetected
	        OR #iqUDT_EquipmentControl.Command.ResetData
	    THEN
	        "FC_Statistics"(ix_Reset := #iqUDT_EquipmentControl.Command.ResetData,
	                        ix_Activate := #iqx_MissingSlatDetected,
	                        ix_RTrigActivate := #sR_TRIG_MissingSlatDetected.Q,
	                        iqUDT_Statistics := #iqUDT_Statistics);

	    END_IF;

	END_REGION


END_FUNCTION_BLOCK

TYPE "UDT_SorterConveyorConfiguration"
TITLE = UDT_SorterConveyorConfiguration
VERSION : 0.1
//User-defined structure of  sorter conveyor parameters.
   STRUCT
      Common : "UDT_ConveyorCommonConfiguration";   // Common configuration
      Forward_Direction : Struct   // Forward Direction configuration
         EnergySaveLenght : DInt;   // Distance conveyor travelled before energy save activate [cm]
         PEC_EoSDistanceOffset : DInt;   // Distance offset between photo eye and the end of conveyor [mm]
         FirstConveyorToStart { ExternalAccessible := 'False'; ExternalVisible := 'False'; ExternalWritable := 'False'} : Bool;   // First conveyor to start cascade mode forward direction
      END_STRUCT;
      CascadeTimeOnDelay : UDInt;   // Cascade time on delay [ms]
      SpeedSetpointPendantLow : Int;   // Extra gap to recovery die back [cm]
      SpeedSetpointLow : Int;   // Low speed setpoint [mm/s]
      SpeedSetpointNominal : Int;   // Nominal speed setpoint [mm/s]
      RTR_at_Speed { ExternalAccessible := 'False'; ExternalVisible := 'False'; ExternalWritable := 'False'} : Bool;   // TRUE = RTR to upstream when sorter reached nominal speed
      Energy { ExternalAccessible := 'False'; ExternalVisible := 'False'; ExternalWritable := 'False'} : Bool;   // Energy save mode enable
   END_STRUCT;

END_TYPE

TYPE "UDT_SpiralVeyorStatus"
VERSION : 0.1
   STRUCT
      MissingSlat { ExternalAccessible := 'False'; ExternalVisible := 'False'; ExternalWritable := 'False'} : Bool;   // Missing slat detected in SpiralVeyor lane
      BrokenChain { ExternalAccessible := 'False'; ExternalVisible := 'False'; ExternalWritable := 'False'} : Bool;   // Broken chain detected in SpiralVeyor lane
      ChainOverlength { ExternalAccessible := 'False'; ExternalVisible := 'False'; ExternalWritable := 'False'} : Bool;   // Warning chain overlength detected in SpiralVeyor lane
   END_STRUCT;

END_TYPE

TYPE "UDT_PendantVT100Interface"
TITLE = Configuation variables for VT100 Radio Pendant
VERSION : 0.1
   STRUCT
      LowSpeedSelected { ExternalAccessible := 'False'; ExternalVisible := 'False'; ExternalWritable := 'False'} : Bool;   // Lowest Speed
      ManualSpeedSelected { ExternalAccessible := 'False'; ExternalVisible := 'False'; ExternalWritable := 'False'} : Bool;   // Manual Speed
      CmdRun { ExternalAccessible := 'False'; ExternalVisible := 'False'; ExternalWritable := 'False'} : Bool;   // Comman to run VFD
      CmdDivert { ExternalAccessible := 'False'; ExternalVisible := 'False'; ExternalWritable := 'False'} : Bool;   // Command to divert
      ServiceModeEngaged { ExternalAccessible := 'False'; ExternalVisible := 'False'; ExternalWritable := 'False'} : Bool;   // Pendant service mode is engaged
      PendantStopHealthy { ExternalAccessible := 'False'; ExternalVisible := 'False'; ExternalWritable := 'False'} : Bool;   // Pedant Stop button is healthy
      PendantReset { ExternalAccessible := 'False'; ExternalVisible := 'False'; ExternalWritable := 'False'} : Bool;   // Reset command from pendant
      RequestSTO { ExternalAccessible := 'False'; ExternalVisible := 'False'; ExternalWritable := 'False'} : Bool;   // Request STO command to safety program
      ForceLowSpeed { ExternalAccessible := 'False'; ExternalVisible := 'False'; ExternalWritable := 'False'} : Bool;   // Force low speed for pin detection
   END_STRUCT;

END_TYPE

TYPE "UDT_SpiralVeyorStatistics"
VERSION : 0.1
   STRUCT
      MissingSlat { S7_SetPoint := 'False'} : "UDT_EventStatistic";   // Statistics of missing slat event
      BrokenChain { S7_SetPoint := 'False'} : "UDT_EventStatistic";   // Statistics of broken chain event
      ChainOverlength { S7_SetPoint := 'False'} : "UDT_EventStatistic";   // Statistics of chain overlength event
   END_STRUCT;

END_TYPE

TYPE "UDT_ConveyorStatistics"
TITLE = UDT_ConveyorStatistics
VERSION : 0.1
//User-defined structure of FB_Conveyor function block statistics.
   STRUCT
      EnergySave : "UDT_EventStatistic";   // Number of times that save energy mode occurs
      ConveyorUp : "UDT_EventStatistic";   // Conveyor up statistics
      ConveyorDown : "UDT_EventStatistic";   // Conveyor down statistics
      ConveyorStop : "UDT_EventStatistic";   // Conveyor down statistics
   END_STRUCT;

END_TYPE

FUNCTION_BLOCK "FB_Displacement"
TITLE = FB_Displacement
{ S7_Optimized_Access := 'TRUE' }
AUTHOR : MHSE
FAMILY : GeneralSystemFunctions
VERSION : 3.0
//Function block to calculate the displacement.
   VAR_IN_OUT
      iqUDT_ConveyorInterface : "UDT_ConveyorInterface";   // Conveyor interface structure Motor
   END_VAR

   VAR
      slr_FormDisplacement { ExternalAccessible := 'False'; ExternalVisible := 'False'; ExternalWritable := 'False'} : LReal;   // Conveyor displacement [cm]
      slr_Correction { ExternalAccessible := 'False'; ExternalVisible := 'False'; ExternalWritable := 'False'} : LReal;   // Correction [cm]
      sx_PositionModeActive { ExternalAccessible := 'False'; ExternalVisible := 'False'; ExternalWritable := 'False'} : Bool;   // Position Mode is used, Will reset after power change
   END_VAR

   VAR_TEMP
      ti_Displacement : Int;   // Conveyor displacement [cm]
   END_VAR

   VAR CONSTANT
      ci_IntMin : Int := -32768;
      ci_IntMax : Int := 32767;
   END_VAR


BEGIN
	(*
	----------------------------------------------------------------------------------------

	Version history:
	Date        | Version   | Author        | Remark
	----------------------------------------------------------------------------------------
	24/05/2019  | 0.1       | L.Klar        | first release MHS TIA 15.1
	24/07/2019  | 2.0       | L.Klar        | 2.0 MHS library release TIA 15.1
	12/09/2019  | 2.1       | P.Majka       | Comments updataed
	04/11/2019  | 2.2       | L.Klar        | Prevoius cycle scan changed from memory to DB variable
	12/11/2019  | 3.0       | P.Majka       | 3.0 MHS library release TIA 15.1
	21/02/2023  | 4.0       | F.Baten       | 4.0 Release TIA 17.5
	31/05/2024  | 4.1       | I.Ajram       | Added Displacement from Position feedback
	*)
	REGION 0 - Mode detection
	    IF #iqUDT_ConveyorInterface.DeltaPosition <> 0 THEN
	        #sx_PositionModeActive := true;
	    END_IF;
	END_REGION


	REGION 1 - Displacement From Speed
	    IF NOT #sx_PositionModeActive THEN
	        REGION 1.1 Calculate Displacement
	            // Displacement is calculated using actual conveyor speed and the previous PLC cycle scan time
	            #slr_FormDisplacement := INT_TO_LREAL(#iqUDT_ConveyorInterface.ActualSpeed) * "DB_Memory".PrevCycleTime / 10000.0;

	            // Correction is used to accumulate the rest of the calculated value
	            #slr_Correction := FRAC(#slr_FormDisplacement) + #slr_Correction;

	            // The actual displacement is a sum of complete parts of the displacement and correction variables
	            #ti_Displacement := DINT_TO_INT(TRUNC(#slr_FormDisplacement) + TRUNC(#slr_Correction));

	        END_REGION

	        REGION 1.2 - Correction check

	            // Correction incrementation or decremantation if it exceeds 1 or -1 in case of negative speed
	            IF (#slr_Correction >= 1)
	            THEN

	                #slr_Correction -= 1;

	            ELSIF (#slr_Correction <= -1)
	            THEN

	                #slr_Correction += 1;

	            END_IF;

	        END_REGION

	        #iqUDT_ConveyorInterface.Displacement := #ti_Displacement;
	    END_IF;
	END_REGION

	REGION 2 - Displacement from Position
	    // pass position displacement from Servo Feedback
	    IF #sx_PositionModeActive THEN
	        #iqUDT_ConveyorInterface.Displacement := #iqUDT_ConveyorInterface.DeltaPosition;

	    END_IF;

	END_REGION
END_FUNCTION_BLOCK

TYPE "UDT_RIOVSUStatus"
VERSION : 0.1
   STRUCT
      PNSlaveNotOnline { ExternalAccessible := 'False'; ExternalVisible := 'False'; ExternalWritable := 'False'} : Bool;   // Profinet slave is not online
      PNSlaveError { ExternalAccessible := 'False'; ExternalVisible := 'False'; ExternalWritable := 'False'} : Bool;   // Profinet slave has an error
      "400VCircuitBreaker" { ExternalAccessible := 'False'; ExternalVisible := 'False'; ExternalWritable := 'False'} : Bool;   // 400V Circuit breaker has tripped
      BrakeCircuitBreaker { ExternalAccessible := 'False'; ExternalVisible := 'False'; ExternalWritable := 'False'} : Bool;   // Brake Circuit breaker has tripped
      BrakeThermalError { ExternalAccessible := 'False'; ExternalVisible := 'False'; ExternalWritable := 'False'} : Bool;   // Brake of the servo unit is giving a thermal error
      "24VPowersupplyError" { ExternalAccessible := 'False'; ExternalVisible := 'False'; ExternalWritable := 'False'} : Bool;   // 24V power supply is in error
      ET200sp_ErrorModule : Array[0..31] of Bool;   // True = ET200sp Module has an error or is offline
      PNSlaveWarning { ExternalAccessible := 'False'; ExternalVisible := 'False'; ExternalWritable := 'False'} : Bool;   // Profinet slave has a warning
   END_STRUCT;

END_TYPE

TYPE "UDT_RIOVSUStatistics"
TITLE = UDT_RIOStatistics
VERSION : 0.1
//User-defined structure of FB_RIO function block statistics.
   STRUCT
      Int400VCBError : "UDT_EventStatistic";   // Statistics of internal 400V circuit breaker not OK
      Ext400VError : "UDT_EventStatistic";   // Statistics of external 400V not OK
      "24VError" : "UDT_EventStatistic";   // Statistics of external 24V not OK
      BrakeCBerror : "UDT_EventStatistic";   // Statistics of brake circuit breaker not OK
      BrakeThermError : "UDT_EventStatistic";   // Statistics of brake thermal error
      PNSlaveNotOnline : "UDT_EventStatistic";   // Statistics of Profinet slave not online
      PNSlaveError : "UDT_EventStatistic";   // Statistics of a Profinet slave error
   END_STRUCT;

END_TYPE

FUNCTION_BLOCK "FB_RIO"
TITLE = FB_RIO
{ S7_Optimized_Access := 'TRUE' }
AUTHOR : MHSE
FAMILY : GeneralSystemFunctions
VERSION : 3.0
// ATTRIBUTES
// AUTO_NUMBER = True
// BLOCK_NUMBER = 225
// END_ATTRIBUTES
//Function block to diagnose remote IO module.
   VAR_INPUT
      is_ET200spPNDeviceName { ExternalAccessible := 'False'; ExternalVisible := 'False'; ExternalWritable := 'False'} : String;   //  Name of the ET200sp device
      ix_24VOk { ExternalAccessible := 'False'; ExternalVisible := 'False'; ExternalWritable := 'False'} : Bool;   //  TRUE when 24VDC is healthy
      ix_SimulationModeActive { ExternalAccessible := 'False'; ExternalVisible := 'False'; ExternalWritable := 'False'} : Bool;   //  TRUE when simulation mode active
      ix_HardwareOk { ExternalAccessible := 'False'; ExternalVisible := 'False'; ExternalWritable := 'False'} : Bool;   //  TRUE when  hardware is Ok
   END_VAR

   VAR_OUTPUT
      qUDT_HMIStatus { ExternalAccessible := 'False'; ExternalVisible := 'False'; ExternalWritable := 'False'} : "UDT_RIOStatus";   //  HMI status structure
      qUDT_Status { ExternalAccessible := 'False'; ExternalVisible := 'False'; ExternalWritable := 'False'} : "UDT_CommonStatus";   //  Common status structure
      qx_PNDeviceOk { ExternalAccessible := 'False'; ExternalVisible := 'False'; ExternalWritable := 'False'} : Bool;   //  Device ok
   END_VAR

   VAR_IN_OUT
      iqUDT_EquipmentControl : "UDT_EquipmentControl";   //  Equipment control structure
      iqUDT_Statistics : "UDT_RIOStatistics";   //  Statistics structure
   END_VAR

   VAR
      sUDT_CommonStatus { ExternalAccessible := 'False'; ExternalVisible := 'False'; ExternalWritable := 'False'; S7_SetPoint := 'False'} : "UDT_CommonStatus";   //  Common status structure
      sUDT_CommonStatusOld { ExternalAccessible := 'False'; ExternalVisible := 'False'; ExternalWritable := 'False'; S7_SetPoint := 'False'} : "UDT_CommonStatus";   //  Common status structure
      sUDT_HMIStatus { ExternalAccessible := 'False'; ExternalVisible := 'False'; ExternalWritable := 'False'; S7_SetPoint := 'False'} : "UDT_RIOStatus";   //  HMI status structure
      sUDT_PNDevice { ExternalAccessible := 'False'; ExternalVisible := 'False'; ExternalWritable := 'False'; S7_SetPoint := 'False'} : "UDT_PNDevice";   //  PN device info structure
      sa_PNPortsStatus { ExternalAccessible := 'False'; ExternalVisible := 'False'; ExternalWritable := 'False'} : Array[1..8] of Bool;   // TRUE when specific port has an error
      sFB_TimerOnOffDelayCheckSupply { ExternalAccessible := 'False'; ExternalVisible := 'False'; ExternalWritable := 'False'; S7_SetPoint := 'False'} : "FB_TimerOnOffDelay";   //  MHS "TimerOnOffDelay" - to delay time for VFD supply contactor
      sR_TRIG_PNSlaveNotOnline {InstructionName := 'R_TRIG'; LibVersion := '1.0'; ExternalAccessible := 'False'; ExternalVisible := 'False'; ExternalWritable := 'False'; S7_SetPoint := 'False'} : R_TRIG;   //  Rising edge for trigger Profinet slave not online statistics
      sR_TRIG_DeviceFound {InstructionName := 'R_TRIG'; LibVersion := '1.0'; ExternalAccessible := 'False'; ExternalVisible := 'False'; ExternalWritable := 'False'; S7_SetPoint := 'False'} : R_TRIG;   //  Rising edge for trigger scan modules
      sR_TRIG_PNSlaveError {InstructionName := 'R_TRIG'; LibVersion := '1.0'; ExternalAccessible := 'False'; ExternalVisible := 'False'; ExternalWritable := 'False'; S7_SetPoint := 'False'} : R_TRIG;   //  Rising edge for trigger Profinet slave error statistics
      si_ModuleStateReturn { ExternalAccessible := 'False'; ExternalVisible := 'False'; ExternalWritable := 'False'} : Int;   //  Status structure
      si_NrOfModulesWithError { ExternalAccessible := 'False'; ExternalVisible := 'False'; ExternalWritable := 'False'} : Int;   //  Number of the faulty modules
      sx_PowerOk { ExternalAccessible := 'False'; ExternalVisible := 'False'; ExternalWritable := 'False'} : Bool;   //  True = External Power OK
      sx_PNSlaveOnline { ExternalAccessible := 'False'; ExternalVisible := 'False'; ExternalWritable := 'False'} : Bool;   //  Profinet device is online and error free
      sx_ConfigurationError { ExternalAccessible := 'False'; ExternalVisible := 'False'; ExternalWritable := 'False'} : Bool;   //  Commissioning: configuration error
   END_VAR

   VAR_TEMP
      ta_Configured : Array[0..127] of Bool;   //  Configured modules array
      ta_Exist : Array[0..127] of Bool;   //  Existing modules array
      ta_Error : Array[0..127] of Bool;   //  Faulty modules array
      ti_NrOfModule : Int;   //  Number of current module
      ti_DiagArraySize : Int;   //  Diagnostic array size
   END_VAR

   VAR CONSTANT
      cui_ConfiguredModulesMode : UInt := 1;   //  Mode selector: 1 = Configured modules scan mode
      cui_ModuleErrorMode : UInt := 2;   //  Mode selector: 2 = Existing modules scan mode
      cui_ExistingModulesMode : UInt := 4;   //  Mode selector: 3 = Module Error scan mode
      ci_PowerSupplyDelayTime : UInt := 4000;   //  Power supply delay time
      ci_NumberOfProfinetPorts : Int := 2;   // Number of Profinet ports in device
   END_VAR


BEGIN
	(*
	----------------------------------------------------------------------------------------

	Version history:
	Date        | Version   | Author        | Remark
	----------------------------------------------------------------------------------------
	24/05/2019  | 0.1       | K.Pokorski    | first release MHS TIA 15.1
	14/06/2019  | 0.2       | K.Pokorski    | Delete trigger in faults reset - Region 4
	14/06/2019  | 0.3       | A.Nowak       | Replacement of instruction if for direct write into variable - Region 3
	24/06/2019  | 0.3       | L.Klar        | Status running added
	19/07/2019  | 0.5       | L.Klar        | Status handling changed, output qx_DeviceOk added
	24/07/2019  | 2.0       | L.Klar        | 2.0 MHS library release TIA 15.1
	14/08/2019  | 2.1       | K.Pokorski    | Profinet number search automatically
	03/09/2019  | 2.2       | TVB           | Updated code for status and statistics, added 24v input to set errors
	09/09/2019  | 2.3       | K.Pokorski    | Updated code for reset errors, changed conditions to start scan loop
	01/10/2019  | 2.4       | K.Pokorski    | Changed region 1 contents to FC
	01/10/2019  | 2.5       | K.Pokorski    | Common status added
	14/10/2019  | 2.6       | L.Klar        | Updated status structure
	14-10-2019  | 2.7       | S. Deulkar    | Created saperate network for status
	12/11/2019  | 3.0       | P.Majka       | 3.0 MHS library release TIA 15.1
	04/11/2019  | 3.1       | F.Baten       | Region 3: ix_SimulationModeActive rearranged to correct position
	08/07/2019  | 3.2       | S.Theocharis  | Write q_Status in every scan. Initialize static status
	09/07/2019  | 3.3       | S.Theocharis  | Initialize the #si_NrOfModulesWithError on the reset
	03/11/2020  | 3.4       | K.Pokorski    | Profinet ports diagnostics added
	02/08/2021  | 3.5       | S. Deulkar    | Added logic to reset error when 24V is not okay.
	21/02/2023  | 4.0       | F.Baten       | 4.0 Release TIA 17.5
	*)

	REGION 1 - Get Device Profinet information

	    "FC_GetDevicePN"(is_PNDeviceName := #is_ET200spPNDeviceName,
	                     ix_SimulationModeActive := #ix_SimulationModeActive,
	                     iqUDT_PND := #sUDT_PNDevice);


	    "FC_GetPNPortStatus"(ii_NumberOfPorts := #ci_NumberOfProfinetPorts,
	                         iUDT_DevicePNInfo := #sUDT_PNDevice,
	                         qa_PortFault => #sa_PNPortsStatus);

	END_REGION

	REGION 2 - Reset errors

	    // reset Profinet Slave error/not online
	    IF #iqUDT_EquipmentControl.Command.Reset
	        OR NOT #ix_24VOk
	    THEN
	        #sUDT_HMIStatus.Specific.PNSlaveNotOnline := FALSE;
	        #sUDT_HMIStatus.Specific.PNSlaveError := FALSE;
	        #sUDT_HMIStatus.Specific.PNSlaveWarning := FALSE;
	        #si_NrOfModulesWithError := 0;
	    END_IF;

	    // reset ET200sp module error status
	    IF #sUDT_HMIStatus.Specific.PNSlaveNotOnline OR #iqUDT_EquipmentControl.Command.Reset OR NOT #ix_24VOk
	    THEN
	        FILL_BLK(IN := FALSE,
	                 COUNT := 32,
	                 OUT => #sUDT_HMIStatus.Specific.ET200sp_ErrorModule[0]);
	    END_IF;

	END_REGION

	REGION 3 - Update PN slave device status
	    // Hardware will only be available after the delay, so the device has time for the initialisation
	    #sFB_TimerOnOffDelayCheckSupply(iudi_OnDelayTime := #ci_PowerSupplyDelayTime,
	                                    ix_SignalToDelay := #ix_24VOk,
	                                    qx_DelayedSignal => #sx_PowerOk);

	    // check if PN device is online
	    IF NOT "DB_ProfinetDiagnostic".ProfinetNetworks[#sUDT_PNDevice.PNNetworknumber].DeviceStatus[#sUDT_PNDevice.PNDeviceNumber].DeviceState.Exist
	        AND #sx_PowerOk
	        OR NOT #sUDT_PNDevice.PNDeviceFound
	        AND NOT #ix_SimulationModeActive
	    THEN

	        #sUDT_HMIStatus.Specific.PNSlaveNotOnline := TRUE;

	    END_IF;

	    // Check if PN ports are healthy
	    IF #sa_PNPortsStatus[1] XOR #sa_PNPortsStatus[2] THEN
	        #sUDT_HMIStatus.Specific.PNSlaveWarning := TRUE;
	    END_IF;


	    // check if PN device has an error
	    IF "DB_ProfinetDiagnostic".ProfinetNetworks[#sUDT_PNDevice.PNNetworknumber].DeviceStatus[#sUDT_PNDevice.PNDeviceNumber].DeviceState.Error
	        AND #sx_PowerOk
	        AND NOT #ix_SimulationModeActive
	        AND NOT #sUDT_HMIStatus.Specific.PNSlaveWarning
	    THEN
	        #sUDT_HMIStatus.Specific.PNSlaveError := TRUE;
	    END_IF;

	    // set bit when PN device is healthy (online and no error)
	    #sx_PNSlaveOnline := NOT #sUDT_HMIStatus.Specific.PNSlaveNotOnline
	    AND #sUDT_PNDevice.PNDeviceFound
	    AND #sx_PowerOk;

	    // create rising edge to scan module status when device is found
	    #sR_TRIG_DeviceFound(CLK := #sUDT_PNDevice.PNDeviceFound);

	END_REGION

	REGION 4 - Status update modules ET200sp
	    // update ET200sp module status
	    IF (#sx_PNSlaveOnline
	        AND (#sUDT_HMIStatus.Specific.PNSlaveError OR
	        #sUDT_HMIStatus.Specific.PNSlaveWarning))
	        OR #sR_TRIG_DeviceFound.Q
	    THEN
	        // get configured modules
	        #si_ModuleStateReturn := ModuleStates(LADDR := "DB_ProfinetDiagnostic".ProfinetNetworks[#sUDT_PNDevice.PNNetworknumber].DeviceStatus[#sUDT_PNDevice.PNDeviceNumber].DeviceState.HW_ID,
	                                              MODE := #cui_ConfiguredModulesMode,
	                                              STATE := #ta_Configured);

	        // get module online status
	        #si_ModuleStateReturn := ModuleStates(LADDR := "DB_ProfinetDiagnostic".ProfinetNetworks[#sUDT_PNDevice.PNNetworknumber].DeviceStatus[#sUDT_PNDevice.PNDeviceNumber].DeviceState.HW_ID,
	                                              MODE := #cui_ExistingModulesMode,
	                                              STATE := #ta_Exist);

	        // get module error status
	        #si_ModuleStateReturn := ModuleStates(LADDR := "DB_ProfinetDiagnostic".ProfinetNetworks[#sUDT_PNDevice.PNNetworknumber].DeviceStatus[#sUDT_PNDevice.PNDeviceNumber].DeviceState.HW_ID,
	                                              MODE := #cui_ModuleErrorMode,
	                                              STATE := #ta_Error);

	        // Handle ET200sp module errors/offline
	        IF (#si_ModuleStateReturn = 0)
	        THEN
	            #si_NrOfModulesWithError := 0;

	            #ti_DiagArraySize := "FC_GetNrOfArrayEl"(iv_Array := "DB_ProfinetDiagnostic".ProfinetNetworks[#sUDT_PNDevice.PNNetworknumber].DeviceStatus[#sUDT_PNDevice.PNDeviceNumber].Module);

	            FOR #ti_NrOfModule := 0 TO (#ti_DiagArraySize - 1) DO

	                // check if the module is configured
	                IF (#ta_Configured[#ti_NrOfModule])
	                THEN
	                    "DB_ProfinetDiagnostic".ProfinetNetworks[#sUDT_PNDevice.PNNetworknumber].DeviceStatus[#sUDT_PNDevice.PNDeviceNumber].Module[#ti_NrOfModule].Configured := TRUE;
	                    // and check if the module is online
	                    IF (#ta_Exist[#ti_NrOfModule])
	                    THEN
	                        "DB_ProfinetDiagnostic".ProfinetNetworks[#sUDT_PNDevice.PNNetworknumber].DeviceStatus[#sUDT_PNDevice.PNDeviceNumber].Module[#ti_NrOfModule].Exist := TRUE;

	                    ELSE
	                        "DB_ProfinetDiagnostic".ProfinetNetworks[#sUDT_PNDevice.PNNetworknumber].DeviceStatus[#sUDT_PNDevice.PNDeviceNumber].Module[#ti_NrOfModule].Exist := FALSE;
	                        #sUDT_HMIStatus.Specific.ET200sp_ErrorModule[#ti_NrOfModule] := TRUE;
	                        // count number of modules with error/offline
	                        #si_NrOfModulesWithError += 1;
	                    END_IF;

	                    // and check if the module has an error
	                    IF (NOT #ta_Error[#ti_NrOfModule])
	                    THEN
	                        "DB_ProfinetDiagnostic".ProfinetNetworks[#sUDT_PNDevice.PNNetworknumber].DeviceStatus[#sUDT_PNDevice.PNDeviceNumber].Module[#ti_NrOfModule].Error := FALSE;

	                    ELSE
	                        "DB_ProfinetDiagnostic".ProfinetNetworks[#sUDT_PNDevice.PNNetworknumber].DeviceStatus[#sUDT_PNDevice.PNDeviceNumber].Module[#ti_NrOfModule].Error := TRUE;
	                        #sUDT_HMIStatus.Specific.ET200sp_ErrorModule[#ti_NrOfModule] := TRUE;
	                        // count number OF modules with error/offline
	                        #si_NrOfModulesWithError += 1;
	                    END_IF;

	                ELSE
	                    // reset module status when module is not configured
	                    "DB_ProfinetDiagnostic".ProfinetNetworks[#sUDT_PNDevice.PNNetworknumber].DeviceStatus[#sUDT_PNDevice.PNDeviceNumber].Module[#ti_NrOfModule].Configured := FALSE;
	                    "DB_ProfinetDiagnostic".ProfinetNetworks[#sUDT_PNDevice.PNNetworknumber].DeviceStatus[#sUDT_PNDevice.PNDeviceNumber].Module[#ti_NrOfModule].Exist := FALSE;
	                    "DB_ProfinetDiagnostic".ProfinetNetworks[#sUDT_PNDevice.PNNetworknumber].DeviceStatus[#sUDT_PNDevice.PNDeviceNumber].Module[#ti_NrOfModule].Error := FALSE;

	                END_IF;
	            END_FOR;
	        END_IF;
	    END_IF;

	END_REGION

	REGION 5 - Check RIO Panel Status
	    // check if PN device is healthy
	    #qx_PNDeviceOk := (#si_NrOfModulesWithError = 0)
	    AND NOT #sUDT_HMIStatus.Specific.PNSlaveNotOnline
	    AND NOT #sUDT_HMIStatus.Specific.PNSlaveError;

	    // set config not ok bit if no device found
	    #sx_ConfigurationError := NOT #sUDT_PNDevice.PNDeviceFound;


	END_REGION

	REGION 6 - Statistics
	    // create trigger on error and create statistics for profinet slave not online
	    #sR_TRIG_PNSlaveNotOnline(CLK := #sUDT_HMIStatus.Specific.PNSlaveNotOnline);

	    IF #iqUDT_EquipmentControl.Command.ResetData OR #sUDT_HMIStatus.Specific.PNSlaveNotOnline
	    THEN

	        "FC_Statistics"(ix_Reset := #iqUDT_EquipmentControl.Command.ResetData,
	                        ix_Activate := #sUDT_HMIStatus.Specific.PNSlaveNotOnline,
	                        ix_RTrigActivate := #sR_TRIG_PNSlaveNotOnline.Q,
	                        iqUDT_Statistics := #iqUDT_Statistics.PNSlaveNotOnline);
	    END_IF;

	    // create trigger on error and create statistics for profinet slave error
	    #sR_TRIG_PNSlaveError(CLK := #sUDT_HMIStatus.Specific.PNSlaveError);

	    IF #iqUDT_EquipmentControl.Command.ResetData OR #sUDT_HMIStatus.Specific.PNSlaveError
	    THEN

	        "FC_Statistics"(ix_Reset := #iqUDT_EquipmentControl.Command.ResetData,
	                        ix_Activate := #sUDT_HMIStatus.Specific.PNSlaveError,
	                        ix_RTrigActivate := #sR_TRIG_PNSlaveError.Q,
	                        iqUDT_Statistics := #iqUDT_Statistics.PNSlaveError);
	    END_IF;

	END_REGION

	REGION 7 - Status

	    #sUDT_CommonStatus.Error := #sUDT_HMIStatus.Specific.PNSlaveError
	    OR #sUDT_HMIStatus.Specific.PNSlaveNotOnline
	    OR #si_NrOfModulesWithError <> 0;

	    // HMI status update
	    IF #sUDT_CommonStatusOld <> #sUDT_CommonStatus                    // update on change
	    THEN

	        // HMI status initialization
	        #sUDT_HMIStatus.Status := 0;

	        // HMI status calculation
	        IF #si_NrOfModulesWithError <> 0                                // Hardware error
	        THEN

	            #sUDT_HMIStatus.Status := "DB_HMIStatusConfiguration".HardwareError;

	        END_IF;

	        IF #sUDT_HMIStatus.Specific.PNSlaveError                       // Profinet error
	            OR #sUDT_HMIStatus.Specific.PNSlaveNotOnline
	        THEN

	            #sUDT_HMIStatus.Status := "DB_HMIStatusConfiguration".ProfinetError;

	        END_IF;
	        #qUDT_Status := #sUDT_CommonStatus;                       // Copy status to output
	        #qUDT_HMIStatus := #sUDT_HMIStatus;                       // Copy HMI status to output
	        #sUDT_CommonStatusOld := #sUDT_CommonStatus;              // Copy status to memory


	    END_IF;

	    //Write status in every scan. AST 8/7/20
	    #qUDT_HMIStatus := #sUDT_HMIStatus;                       // Copy HMI status to output

	END_REGION

	REGION 8 - Report to control block

	    // Function to manage report between control block and conveyor block
	    "FC_EquipmentReport"(iUDT_Status := #sUDT_CommonStatus,
	                         iqUDT_Control := #iqUDT_EquipmentControl);

	END_REGION

END_FUNCTION_BLOCK

TYPE "UDT_VSUInterface"
TITLE = UDT_VSUInterface
VERSION : 0.1
//User-defined structure of VSU interface parameters.
   STRUCT
      Decisionpoint : Int;   // Point in tracking where the destination is found on the VSU conveyor [mm]
      RequestedPosition : Int;   // Position Requested by destination block
      PositionSetpoint : Int;   // Position number (as configured) to go to by positioning device
      PositionActual : Int;   // Position number the positioning device is actually on
      SwitchingTime : UInt;   // Time it takes to go from one position to the next [ms]
      VSUMainPowerOk { ExternalAccessible := 'False'; ExternalVisible := 'False'; ExternalWritable := 'False'} : Bool;   // True = Main power for VSU ok
      BrakeOk { ExternalAccessible := 'False'; ExternalVisible := 'False'; ExternalWritable := 'False'} : Bool;   // True = VSU brake is ok
      PNDeviceOk { ExternalAccessible := 'False'; ExternalVisible := 'False'; ExternalWritable := 'False'} : Bool;   // Device ok
      Automatic { ExternalAccessible := 'False'; ExternalVisible := 'False'; ExternalWritable := 'False'} : Bool;   // Automatic mode request
      RunEnabled { ExternalAccessible := 'False'; ExternalVisible := 'False'; ExternalWritable := 'False'} : Bool;   // Running of the positioning device is enabled by VSU
      GoReference { ExternalAccessible := 'False'; ExternalVisible := 'False'; ExternalWritable := 'False'} : Bool;   // Activate reference run by VSU
      Referenced { ExternalAccessible := 'False'; ExternalVisible := 'False'; ExternalWritable := 'False'} : Bool;   // Positioning device is referenced
      Manual { ExternalAccessible := 'False'; ExternalVisible := 'False'; ExternalWritable := 'False'} : Bool;   // Manual mode request
      Reference_command { ExternalAccessible := 'False'; ExternalVisible := 'False'; ExternalWritable := 'False'} : Bool;   // Refference command
      JogUp { ExternalAccessible := 'False'; ExternalVisible := 'False'; ExternalWritable := 'False'} : Bool;   // Jog request to move equipment up
      JogDown { ExternalAccessible := 'False'; ExternalVisible := 'False'; ExternalWritable := 'False'} : Bool;   // Jog request to move equipment down
      Ready { ExternalAccessible := 'False'; ExternalVisible := 'False'; ExternalWritable := 'False'} : Bool;   // Positioning block is running and error free
      MotorRunning { ExternalAccessible := 'False'; ExternalVisible := 'False'; ExternalWritable := 'False'} : Bool;   // Motor is running
      Positioning { ExternalAccessible := 'False'; ExternalVisible := 'False'; ExternalWritable := 'False'} : Bool;   // positioning device is moving to its position
      ResetStatistics { ExternalAccessible := 'False'; ExternalVisible := 'False'; ExternalWritable := 'False'} : Bool;   // Reset statistics
      InternalErrorRIOPanel { ExternalAccessible := 'False'; ExternalVisible := 'False'; ExternalWritable := 'False'} : Bool;   // RIO panel has an internal error
      InternalWarningRIOPanel { ExternalAccessible := 'False'; ExternalVisible := 'False'; ExternalWritable := 'False'} : Bool;   // RIO panel has an internal waring
      InternalErrorVFD { ExternalAccessible := 'False'; ExternalVisible := 'False'; ExternalWritable := 'False'} : Bool;   // positioning device internal error
      InternalWarningVFD { ExternalAccessible := 'False'; ExternalVisible := 'False'; ExternalWritable := 'False'} : Bool;   // positioning device has a warning
      InternalErrorReset { ExternalAccessible := 'False'; ExternalVisible := 'False'; ExternalWritable := 'False'} : Bool;   // Reset internal faults
      StartLowSpeed { ExternalAccessible := 'False'; ExternalVisible := 'False'; ExternalWritable := 'False'} : Bool;   // Positioning device starting in low speed
      RequestDieBackUpstream { ExternalAccessible := 'False'; ExternalVisible := 'False'; ExternalWritable := 'False'} : Bool;   // External request die back to the upstream conveyor of the VSU
      ExternalHold { ExternalAccessible := 'False'; ExternalVisible := 'False'; ExternalWritable := 'False'} : Bool;   // External request to stop the VSU conveyor
   END_STRUCT;

END_TYPE

TYPE "UDT_UnloaderCommand"
VERSION : 0.1
   STRUCT
      Disable { ExternalAccessible := 'False'; ExternalVisible := 'False'; ExternalWritable := 'False'} : Bool;   // Disable unloader
   END_STRUCT;

END_TYPE

TYPE "UDT_LoaderCommand"
VERSION : 0.1
   STRUCT
      Disable { ExternalAccessible := 'False'; ExternalVisible := 'False'; ExternalWritable := 'False'} : Bool;   // Disable loader
   END_STRUCT;

END_TYPE

FUNCTION_BLOCK "FB_PEC"
TITLE = FB_PEC
{ S7_Optimized_Access := 'TRUE' }
AUTHOR : MHSE
FAMILY : Conveyor
VERSION : 3.0
// ATTRIBUTES
// AUTO_NUMBER = True
// BLOCK_NUMBER = 219
// END_ATTRIBUTES
   VAR_INPUT
      ix_PEC { ExternalAccessible := 'False'; ExternalVisible := 'False'; ExternalWritable := 'False'} : Bool;   // Signal of the PEC
      iUDT_PECConfiguration { ExternalAccessible := 'False'; ExternalVisible := 'False'; ExternalWritable := 'False'} : "UDT_PECConfiguration";   // PEC configuration structure
   END_VAR

   VAR_OUTPUT
      qx_PECFiltered { ExternalAccessible := 'False'; ExternalVisible := 'False'; ExternalWritable := 'False'} : Bool;   // PEC Filtered
      qUDT_HMIStatus { ExternalAccessible := 'False'; ExternalVisible := 'False'; ExternalWritable := 'False'} : "UDT_PECStatus";   // Status structure
   END_VAR

   VAR_IN_OUT
      iqUDT_ConveyorInterface : "UDT_ConveyorInterface";   // Interface structure
      iqUDT_PECStatistics : "UDT_PECStatistics";   // Statistics structure
   END_VAR

   VAR
      s_Status { ExternalAccessible := 'False'; ExternalVisible := 'False'; ExternalWritable := 'False'; S7_SetPoint := 'False'} : "UDT_PECStatus";   // Status structure
      s_StatusOld { ExternalAccessible := 'False'; ExternalVisible := 'False'; ExternalWritable := 'False'; S7_SetPoint := 'False'} : "UDT_PECStatus";   // Auxiliary status structure
      sx_Enable { ExternalAccessible := 'False'; ExternalVisible := 'False'; ExternalWritable := 'False'} : Bool;   // Enable
   END_VAR
   VAR RETAIN
      si_AuxJamDisplacement { ExternalAccessible := 'False'; ExternalVisible := 'False'; ExternalWritable := 'False'} : Int;   // Auxiliary variable to calculate displacement when PEC is blocked
   END_VAR
   VAR
      sx_PECFiltered { ExternalAccessible := 'False'; ExternalVisible := 'False'; ExternalWritable := 'False'} : Bool;   // Photo eye filtered
      PEC_TimerOnOffDelay { ExternalAccessible := 'False'; ExternalVisible := 'False'; ExternalWritable := 'False'; S7_SetPoint := 'False'} : "FB_TimerOnOffDelay";   // Filtering end of section photo eye signal
      R_TRIG_PECJam {InstructionName := 'R_TRIG'; LibVersion := '1.0'; ExternalAccessible := 'False'; ExternalVisible := 'False'; ExternalWritable := 'False'; S7_SetPoint := 'False'} : R_TRIG;   // Rising edge trigger PEC jam
   END_VAR


BEGIN
	(*
	----------------------------------------------------------------------------------------

	Version history:
	Date        | Version   | Author        | Remark
	----------------------------------------------------------------------------------------
	04/10/2019  | 2.0       | S. Nikodem    | first release TIA 15.1
	09/10/2019  | 2.1       | L.Klar        | Internal PEC error added
	28/10/2019  | 2.2       | S. Nikodem    | Change sign in region 2 - equal to greater then
	29/10/2019  | 2.3       | L.Klar        | UDT_PECStatus output variable changed, interface comments adjusted
	29/10/2019  | 2.4       | L.Klar        | Region 4 - time input corrected
	12/11/2019  | 3.0       | P.Majka       | 3.0 MHS library release TIA 15.1
	26/11/2019  | 3.1       | P.Majka       | Static variable name change to PEC from EOS PEC
	12/12/2019  | 3.2       | C. Leite      | Absolute displacement value to control jam error in both directions
	21/02/2023  | 4.0       | F.Baten       | 4.0 Release TIA 17.5
	12/03/2024  | 4.1       | S. Nieswiec   | Small variable name changes according to current standard
	*)

	REGION 1 - Triggers

	    // Rising edge PEC Jam
	    #R_TRIG_PECJam(CLK := #s_Status.Jam);

	END_REGION

	REGION 2 - Active function

	    // To activate the jam monitoring the jam displacement limit  must be configured up to zero.
	    #sx_Enable := #iUDT_PECConfiguration.JamDisplacementLimit > 0;

	END_REGION

	REGION 3 - Reset errors

	    // Jam error is reset when reset bit is active and jam error is active and is connfigured alllow reset jam with PEC blocked or photo eye is not active
	    IF #iqUDT_ConveyorInterface.InternalErrorReset
	        AND (#iUDT_PECConfiguration.ResetWithPECBlocked
	        OR (NOT #iUDT_PECConfiguration.ResetWithPECBlocked
	        AND #sx_PECFiltered))
	        AND #s_Status.Jam
	    THEN

	        #si_AuxJamDisplacement := 0;
	        #s_Status.Jam := FALSE;

	    END_IF;

	END_REGION

	REGION 4 - Photo eye filters

	    // End of section photo eye signal filter timer
	    #PEC_TimerOnOffDelay(iudi_OnDelayTime := #iUDT_PECConfiguration.TimeOnDelay,
	                         iudi_OffDelayTime := #iUDT_PECConfiguration.TimeOffDelay,
	                         ix_SignalToDelay := #ix_PEC,
	                         ix_Enable := TRUE,
	                         qx_DelayedSignal => #sx_PECFiltered);

	    // Write the current status of the photo eye
	    #s_Status.PEC := #sx_PECFiltered;
	    #qx_PECFiltered := #sx_PECFiltered;

	END_REGION

	REGION 5 - Jam detection

	    IF NOT #sx_PECFiltered                                                    // Photo eye blocked
	        AND #sx_Enable                                                            // Active of checking the PEC jam
	    THEN

	        #si_AuxJamDisplacement += ABS(#iqUDT_ConveyorInterface.Displacement);

	    ELSE

	        #si_AuxJamDisplacement := 0;

	    END_IF;

	    // Compare jam auxiliary counter with displacement jam configured
	    IF #si_AuxJamDisplacement > #iUDT_PECConfiguration.JamDisplacementLimit
	    THEN

	        #s_Status.Jam := TRUE;

	    END_IF;

	END_REGION

	REGION 6 - Statistics

	    // Statistics Jam PEC
	    IF #s_Status.Jam                                                                // PEC jam error active
	        OR #iqUDT_ConveyorInterface.ResetStatistics                                       // Reset statistics
	    THEN

	        "FC_Statistics"(ix_Reset := #iqUDT_ConveyorInterface.ResetStatistics,
	                        ix_Activate := #s_Status.Jam,
	                        ix_RTrigActivate := #R_TRIG_PECJam.Q,
	                        iqUDT_Statistics := #iqUDT_PECStatistics.Jam);

	    END_IF;

	END_REGION

	REGION 7 - Internal PEC error

	    IF #s_Status.Jam
	    THEN

	        #iqUDT_ConveyorInterface.InternalErrorPEC := TRUE;

	    END_IF;

	END_REGION


	REGION 8 - Status

	    // Status update on change
	    IF #s_StatusOld <> #s_Status
	    THEN

	        #qUDT_HMIStatus := #s_Status;
	        #s_StatusOld := #s_Status;

	    END_IF;

	END_REGION
END_FUNCTION_BLOCK

TYPE "UDT_VfdConfiguration"
TITLE = UDT_VFD_Configuration
VERSION : 0.1
//User-defined structure oparameters.
   STRUCT
      GearRatio : Real;   // Gear box value X = turns at input to get 1 turn at output
      ReferenceRPM : Real;   // VFD speed max - reference [rpm]
      WheelEndPerimeter : Real;   // Perimeter of wheel at the end of gear [mm]
      VFDRampUpTime : UDInt;   // VFD ramp up time for monitoring starting [ms]
      VFDRampDownTime : UDInt;   // VFD ramp up time for monitoring stopping [ms]
      SpeedSetpointWindow : Int := 5;   // VFD speed setpoint window (tolerance) [mm/s]
      VFDPNDeviceName : String;   // VFD's Profinet device name
      DirectionReversal { ExternalAccessible := 'False'; ExternalVisible := 'False'; ExternalWritable := 'False'} : Bool;   // If true, direction will be swapped
      InterlockFwd { ExternalAccessible := 'False'; ExternalVisible := 'False'; ExternalWritable := 'False'} : Bool;   // False when turning in forward direction is not possible / allowed
      InterlockRvs { ExternalAccessible := 'False'; ExternalVisible := 'False'; ExternalWritable := 'False'} : Bool;   // False when turning in reverse direction is not possible / allowed
      VFDStartupTime : UDInt := 2000;   // Time when the motor should start [ms]
   END_STRUCT;

END_TYPE

TYPE "UDT_VfdNordPI"
TITLE = UDT_VfdNordPI
VERSION : 0.1
//User-defined structure of VFD Nord input telegram.
   STRUCT
      ZSW : Struct   // Status word
         SetpointReached { ExternalAccessible := 'False'; ExternalVisible := 'False'; ExternalWritable := 'False'} : Bool;   // 0 = Actual value does not corresponf to setpoint. 1 = Actual value matches the setpoint
         BusControlActive { ExternalAccessible := 'False'; ExternalVisible := 'False'; ExternalWritable := 'False'} : Bool;   // 0 = Control on local device active. 1 = The master has beed requestd to take over control
         "StartFunction481.9" { ExternalAccessible := 'False'; ExternalVisible := 'False'; ExternalWritable := 'False'} : Bool;   // 1 = Bus bit 10 of status word is set P481
         RotationRightIsOn { ExternalAccessible := 'False'; ExternalVisible := 'False'; ExternalWritable := 'False'} : Bool;   // 1 = The FI output voltage has a RH rotation field
         RotationLeftIsOn { ExternalAccessible := 'False'; ExternalVisible := 'False'; ExternalWritable := 'False'} : Bool;   // 1 = The FI output voltage has a LH rotation field
         "StartFunction481.10" { ExternalAccessible := 'False'; ExternalVisible := 'False'; ExternalWritable := 'False'} : Bool;   // 1 = Bus bit 13 of status word is set P481
         ParameterSetBit0ON { ExternalAccessible := 'False'; ExternalVisible := 'False'; ExternalWritable := 'False'} : Bool;   // Parameter set bit 0 status
         ParameterSetBit1ON { ExternalAccessible := 'False'; ExternalVisible := 'False'; ExternalWritable := 'False'} : Bool;   // Parameter set bit 0 status
         ReadyToStart { ExternalAccessible := 'False'; ExternalVisible := 'False'; ExternalWritable := 'False'} : Bool;   // 1 = Initialisation completed, charging relay switched on, output voltage disabled
         ReadyForOperation { ExternalAccessible := 'False'; ExternalVisible := 'False'; ExternalWritable := 'False'} : Bool;   // 0 = No switch-on command present or fault. 1 = The inverted can start with the command "Enable operation"
         OperationEnabled { ExternalAccessible := 'False'; ExternalVisible := 'False'; ExternalWritable := 'False'} : Bool;   // 1 = The output voltage is enabled; ramp of the frequency inverter up to the existing setpoint
         Fault : Bool := FALSE;   // 1 = Drive unit defective, not ready for operation
         VoltageEnabled { ExternalAccessible := 'False'; ExternalVisible := 'False'; ExternalWritable := 'False'} : Bool;   // 0 = "Disable voltage" command present
         EmergencyStop { ExternalAccessible := 'False'; ExternalVisible := 'False'; ExternalWritable := 'False'} : Bool;   // 0 = "Emergency stop" command present
         StartingDisabled { ExternalAccessible := 'False'; ExternalVisible := 'False'; ExternalWritable := 'False'} : Bool;   // 1 = With the command "Standby" the FI goes into status "Ready to switch on"
         WarningActive { ExternalAccessible := 'False'; ExternalVisible := 'False'; ExternalWritable := 'False'} : Bool;   // 1 = Drive operation continues, no acknowledgement necessary
      END_STRUCT;
      ActualSpeed : Int;   // Actual calculated speed [rpm]. [Range  -200% ..200%][100%=4000HEX/ 16384DEC = P202 nominal speed]
      FaultCode : Int;   // Actual fault code
   END_STRUCT;

END_TYPE

TYPE "UDT_VfdStatus"
TITLE = UDT_VfdStatus
VERSION : 0.1
//User-defined structure of VFD status.
   STRUCT
      ErrorCode : Int;   // Error code
      SubErrorCode : Int;   // Sub error code
      PNSlaveNotonline : Bool := FALSE;   // Profinet slave is not on line
      PNSlaveError : Bool := FALSE;   // Profinet slave has an error
      InternalError : Bool := FALSE;   // A VFD internal error is active, see error code
      InternalWarning : Bool := FALSE;   // A VFD internal warning is active, see error code
      CommunicationErrorMovikit : Bool := FALSE;   // Communication error with MoviKit
      VFDRunningFeedbackError : Bool := FALSE;   // Motor is not running
      PNSlaveWarning { ExternalAccessible := 'False'; ExternalVisible := 'False'; ExternalWritable := 'False'} : Bool;   // Profinet slave has a warning
   END_STRUCT;

END_TYPE

TYPE "UDT_CaljanStatistics"
TITLE = UDT_UnloaderStatistics
VERSION : 0.1
//User-defined structure of FB_Unloader function block statistics.
   STRUCT
      EnergySave : "UDT_EventStatistic";   // Number of times that save energy mode occurs
      ExtendableUpTime : "UDT_EventStatistic";   // Conveyor up time
      ExtendableDownTime : "UDT_EventStatistic";   // Conveyor down time
      VFDError : "UDT_EventStatistic";   // VFD Error
      NotHealthy : "UDT_EventStatistic";   // Extendable not healthy
      TooLongParcel : "UDT_EventStatistic";   // Too long parcels
      PEC_EOS : "UDT_PECStatistics";   // PEC error
      PNNodeNotOnline : "UDT_EventStatistic";   // PN node not online
      PNNodeError : "UDT_EventStatistic";   // PN node has error
   END_STRUCT;

END_TYPE

TYPE "UDT_VfdNordPO"
TITLE = UDT_VfdNordPO
VERSION : 0.1
//User-defined structure of VFD Nord output telegram.
   STRUCT
      STW : Struct   // Control Word
         "StartFunction408.11" { ExternalAccessible := 'False'; ExternalVisible := 'False'; ExternalWritable := 'False'} : Bool;   // 1 = Bus bit 8 of control word is set. P480
         "StartFunction408.12" { ExternalAccessible := 'False'; ExternalVisible := 'False'; ExternalWritable := 'False'} : Bool;   // 1 = Bus bit 8 of control word is set. P480
         ControlDataValid { ExternalAccessible := 'False'; ExternalVisible := 'False'; ExternalWritable := 'False'} : Bool;   // 1 = The bus master trasnfers valid process data. 0 = The transmitted process data are invalid
         RotationRightOn { ExternalAccessible := 'False'; ExternalVisible := 'False'; ExternalWritable := 'False'} : Bool;   // 1 = Switch on rotation right
         RotationLeftOn { ExternalAccessible := 'False'; ExternalVisible := 'False'; ExternalWritable := 'False'} : Bool;   // 1 = Switch on rotation left
         Reserved { ExternalAccessible := 'False'; ExternalVisible := 'False'; ExternalWritable := 'False'} : Bool;   // Reserved from NORD
         ParameterSetBit0 { ExternalAccessible := 'False'; ExternalVisible := 'False'; ExternalWritable := 'False'} : Bool;   // Activates parameter set
         ParameterSetBit1 { ExternalAccessible := 'False'; ExternalVisible := 'False'; ExternalWritable := 'False'} : Bool;   // Activates parameter set
         ReadyForOperation { ExternalAccessible := 'False'; ExternalVisible := 'False'; ExternalWritable := 'False'} : Bool;   // 1 = Set the frequency inverter to standby. 0=Reverse with brake ramp
         DisableVoltage { ExternalAccessible := 'False'; ExternalVisible := 'False'; ExternalWritable := 'False'} : Bool;   // 0 = Switch off the frequency inverter output voltage. 1 = Cancel "Disable voltage"
         EmergencyStop { ExternalAccessible := 'False'; ExternalVisible := 'False'; ExternalWritable := 'False'} : Bool;   // 0 = Emergency stop with programmed estop time. Not Fail Safe Estop. 1 = Cancel condition "Emergency stop"
         EnableOperation { ExternalAccessible := 'False'; ExternalVisible := 'False'; ExternalWritable := 'False'} : Bool;   // 1 = Enable output voltage acceleration to setpoint. 0 = Block voltage, switch off output voltage
         EnablePulsles { ExternalAccessible := 'False'; ExternalVisible := 'False'; ExternalWritable := 'False'} : Bool;   // 1 = Enable acceleration encoder. 0 = Acceleraton encoder is set to zero
         EnableRamp { ExternalAccessible := 'False'; ExternalVisible := 'False'; ExternalWritable := 'False'} : Bool;   // 1 = Enable setpoint on acceleration encoder. 0 = Freeze the setpoint provided by the acceleration encoder
         EnableSetpoint { ExternalAccessible := 'False'; ExternalVisible := 'False'; ExternalWritable := 'False'} : Bool;   // 1 = Activate the selected setpoint on the acceleration encoder. 0= Set the selected setpoint on the acceleration encoder to 0
         Acknowledge { ExternalAccessible := 'False'; ExternalVisible := 'False'; ExternalWritable := 'False'} : Bool;   // 0-->1 = Inactive errors are acknowledged
      END_STRUCT;
      FrequencySetPoint : Int;   // Frequency HZ SetPoint to VFD 100%=4000HEX /16384 DEC . 0% = 0000HEX / 0 DEC Normalization with P105
      RampTimeSetPoint : Int;   // Ramp time to VFD [Range 0..200%][100% = 4000HEX /16384DEC = 10sec]
   END_STRUCT;

END_TYPE

TYPE "UDT_CommisioningNord"
VERSION : 0.1
   STRUCT
      HWAdress : Int;   // Actual dipswitch adress of the VFD
      i_ParCRC : Word;   // VFD generated CRC
      CommissionError { ExternalAccessible := 'False'; ExternalVisible := 'False'; ExternalWritable := 'False'} : Bool;   // Commissioning error active
   END_STRUCT;

END_TYPE

TYPE "UDT_CaljanCommand"
VERSION : 0.1
   STRUCT
      Disable { ExternalAccessible := 'False'; ExternalVisible := 'False'; ExternalWritable := 'False'} : Bool;   // Disable unloader
   END_STRUCT;

END_TYPE

TYPE "UDT_VfdStatistics"
TITLE = UDT_VFDStatistics_SEW
VERSION : 0.1
//User-defined structure of FB_VFD_SEW_MOVI-C function block statistics.
   STRUCT
      PNSlaveNotOnline : "UDT_EventStatistic";   // Statistics of Profinet slave not online
      PNSlaveError : "UDT_EventStatistic";   // Statistics of a Profinet slave error
      VFDInternalError : "UDT_EventStatistic";   // Statistics of an internal VFD error
      CommunicationErrorMovikit : "UDT_EventStatistic";   // Statistics of a communication error
      Running : "UDT_EventStatistic";   // Statistics for running time
   END_STRUCT;

END_TYPE

FUNCTION_BLOCK "FB_VfdNORDCommissioning"
TITLE = Block for parameterising NORD VFD
{ S7_Optimized_Access := 'TRUE' }
VERSION : 0.1
// ATTRIBUTES
// AUTO_NUMBER = True
// BLOCK_NUMBER = 234
// END_ATTRIBUTES
   VAR_INPUT
      ihw_HardwareID { ExternalAccessible := 'False'; ExternalVisible := 'False'; ExternalWritable := 'False'} : HW_IO := 0;   // Device hardware ID
      iudt_MotorData { ExternalAccessible := 'False'; ExternalVisible := 'False'; ExternalWritable := 'False'} : "UDT_MotorData";
      ir_ReferenceFrequency { ExternalAccessible := 'False'; ExternalVisible := 'False'; ExternalWritable := 'False'} : Real;
      ix_VFDReadyToRun { ExternalAccessible := 'False'; ExternalVisible := 'False'; ExternalWritable := 'False'} : Bool;   // Condition to start motor identyfication
   END_VAR

   VAR_OUTPUT
      qi_HWAdress { ExternalAccessible := 'False'; ExternalVisible := 'False'; ExternalWritable := 'False'} : Int;
      qx_Busy { ExternalAccessible := 'False'; ExternalVisible := 'False'; ExternalWritable := 'False'} : Bool;   // Parametrisation in progress
      qx_Done { ExternalAccessible := 'False'; ExternalVisible := 'False'; ExternalWritable := 'False'} : Bool;   // Parametrisation done
      qx_Error { ExternalAccessible := 'False'; ExternalVisible := 'False'; ExternalWritable := 'False'} : Bool;   // Parametrisation error
      qx_24VCommissioningDone { ExternalAccessible := 'False'; ExternalVisible := 'False'; ExternalWritable := 'False'} : Bool;   // 24V commissioning done succesfully
   END_VAR

   VAR_IN_OUT
      iqx_Enable { ExternalAccessible := 'False'; ExternalVisible := 'False'; ExternalWritable := 'False'} : Bool;   // Input enable signal
   END_VAR

